//Check for next correction update 
IF fCurrentColumnPos + _fColumnsToPrecharge > nChargedColumns AND nChargedColumns <= sDefGridSettings.nGridSizeX THEN
  fCurrentPreCharge := fCurrentColumnPos + _fColumnsToPrecharge;
  IF bEnableDeformation THEN 
    // sync deformation points
    WHILE FLOOR(fCurrentPreCharge) > nChargedColumns AND nChargedColumns <= sDefGridSettings.nGridSizeX DO
      nAvailPoints := _pAttachedCt^.nAvailableGridPoints;
      IF nAvailPoints >= sDefGridSettings.nGridSizeY * (nChargedColumns+1) THEN // Complete column available?
        nAvailPoints_mem := 0;
        LogLvl(Lvl:=E_LogSeverity.Debug, Msg:=F_Concat2('Charge CG col: ',TO_STRING(nChargedColumns)));
        FOR nRow := 0 TO sDefGridSettings.nGridSizeY - 1 DO
          // get points
          IF _pAttachedCt^.getDeformationPoint(nCol:=nChargedColumns, nRow:=nRow, sPoint => sPoint) THEN
            // transfer the displacement into a correction
            sPoint.dx := sPoint.dx;   // nothing to change
            sPoint.dy := sPoint.dy;
            
            // apply PU corrections
            correctionUpdate(pPoint:=ADR(sPoint));
            
            // correction limitation
            correctionLimit(pPoint:=ADR(sPoint));
            
            // send point
            IF NOT fbPs.newGridPoint(sPoint:=sPoint) THEN
               LogError(Msg:='stream new point failed');
               gridUpdate:=FALSE;
               RETURN;
            END_IF
          ELSE
            LogError(Msg:='get new grid point failed');
            gridUpdate:=FALSE;
          END_IF
        END_FOR
        
        nChargedColumns := nChargedColumns + 1;
      ELSE
        IF nAvailPoints > nAvailPoints_mem THEN // log once or after every update of new available poinst
          LogError(Msg:='point column expected but not available');
        END_IF
        nAvailPoints_mem := nAvailPoints;
        gridUpdate:=FALSE;
        RETURN;
      END_IF 
    END_WHILE
  ELSE
    // send points with no deformation
    FOR nRow := 0 TO sDefGridSettings.nGridSizeY - 1 DO
        MEMSET(destAddr:=ADR(sPoint), fillByte:=0, n:=SIZEOF(sPoint));
        sPoint.col := TO_DINT(nChargedColumns);
        sPoint.row := TO_DINT(nRow);
        IF NOT fbPs.newGridPoint(sPoint:=sPoint) THEN
           LogError(Msg:='stream new point failed');
           gridUpdate:=FALSE;
           RETURN;
        END_IF
    END_FOR
    nChargedColumns := nChargedColumns + 1;
  END_IF
END_IF
END_METHOD

METHOD InitWorkerPrint : BOOL
VAR_INPUT
  pAdsPg                : POINTER TO ST_ADS_PG;       // pg ads reference (worker prints ads)
  iDefGridParamMediator : I_ParamMediator;            // for deformation settings
  fLimitCorrectionX     : LREAL;                      // correction limit in y (abs) [px]
  fLimitCorrectionY     : LREAL;                      // correction limit in y (abs) [px]
END_VAR
IF NOT bInitialized            THEN LogError('Base Worker not initialized! call init() before'); RETURN; END_IF
IF pAdspg = 0 THEN LogError('InitWorkerPrint: invalid parameter proviced'); RETURN; END_IF
IF iDefGridParamMediator = 0   THEN bInitialized := FALSE; LogError('Invalid parameter, no valid param mediator'); RETURN; END_IF

// Worker specific init
_pAdsPg := pAdsPg;
_iParamMediator := iDefGridParamMediator;

_fLimitCorrectionX := ABS(fLimitCorrectionX);
_fLimitCorrectionY := ABS(fLimitCorrectionY);

// Print Aggregate
fbPa.bSyncAfterDone := FALSE;
fbPa.init(iPcAdapter := fB_PcAdapter, iPsInterface := fbPs);
END_METHOD

METHOD mJobPause
END_METHOD

METHOD   mJobStart
VAR_INPUT
	sJobDef	: CalmarCompPrint.I_JobDefinition;
END_VAR
// Config workers static variables
_fCtSecurityReleasePos := F_MeterToSubPixel(fPosMeter:=sJobDef.fImageDepth/1000 + fC_MIN_SHEET_GAP, fResoSubPx:=_fPrintResolution*_fSubPxResolution);

IF NOT bWorkerEnable THEN RETURN; END_IF  // only if enabled

fbPa.jobStart();

_sCurrentImgDepth := sJobDef.fImageDepth/1000;
_bEndless := sJobDef.isEndless();

_bJobActive := TRUE;
END_METHOD

METHOD  mJobStop
VAR_INPUT
	sStatus	: CalmarCompPrint.I_JobStatus;
END_VAR
fbPa.jobStop();
_bJobActive := FALSE;
_bPaStarted := FALSE;
_bPaStartRequested := FALSE;
END_METHOD

METHOD mProduced
VAR_INPUT
	(* current progress*)
	sProgress	: CalmarCompPrint.I_JobProgress;
END_VAR
END_METHOD

METHOD RegisterGridCorrection : BOOL
VAR_INPUT
  iGridCorrection : I_GridPointCorrection;
END_VAR
VAR
  i : UDINT;
END_VAR
IF iGridCorrection = 0 THEN LogError('registerGridCorrection: ivalid interface, ignore'); RETURN; END_IF
IF nPointCorrections >= nC_NUM_POINTCORRECTIONS THEN LogError('registerGridCorrection: too many corrections registred, ignore'); RETURN; END_IF

nPointCorrections := nPointCorrections + 1;
iPointCorrections[nPointCorrections] := iGridCorrection;
END_METHOD

METHOD registerPc : BOOL
VAR_INPUT
  iNewPC : I_PC;
END_VAR
registerPc := fB_PcAdapter.registerPc(iNewPC := iNewPC);
END_METHOD

METHOD registerPh : BOOL
VAR_INPUT
    iPH : I_PH;
    iNewCG : I_Correction_Grid;   // correction grid interface
END_VAR
//Attach head to print station
IF iPH <> 0 THEN
  fbPs.registerCG(iNewPh:=iPH, iNewCG:=iNewCG);
END_IF
END_METHOD

METHOD PRIVATE sim
END_METHOD

METHOD PRIVATE updateWorkerPosition
VAR_INPUT
END_VAR
// Update only without attached container
IF _pAttachedCt = 0 THEN RETURN; END_IF

//Start offset update
IF _fPrintStartOffset <> (fPrintStartOffset + _iWorkerParams.fDetectToRefPos) THEN //Worker position changed
  _fPrintStartOffset := fPrintStartOffset + _iWorkerParams.fDetectToRefPos;
END_IF

//Worker position update
IF _fWorkerPosition <> (_fPrintStartOffset + (_fStartShiftOffset + _fStartShiftFactor * fMasterSpeed)) THEN   // Worker position changed (camera settings change)
  // WorkerPosition = PrintStart offset - pre-start offset
  fPosition := _fPrintStartOffset + (_fStartShiftOffset + _fStartShiftFactor * fMasterSpeed);
END_IF
END_METHOD

METHOD  work
VAR
  bDeformErr : BOOL;
  nDeformStep : E_DeformationStep;
END_VAR
IF _iWorkerParams = 0 OR _iParamMediator = 0 THEN F_Report_Error(ErrType:=EN_REPORT_ERROR_TYPE.Report_Error_0Pointer); RETURN; END_IF
bError := FALSE; nError := 0;

updateWorkerPosition();  // calculate and set worker position

SUPER^.work();

(*Print correction*)
fbDropSpeedComp(fMasterSpeed:=fMasterSpeed, fDropTravelDistance:=fPUElevation);


(*Update virtual encoder on all controller boards*)
fB_PcAdapter.setEncoderPos(nPrintPos);
fB_PcAdapter();

(*Call print aggregate*)
rTrigHwSync(CLK:=bHardwareSync); 
IF rTrigHwSync.Q THEN fbPa.sync(); END_IF   // external sync cmd
fbPa.bHold := bHardwareHold;                // external hw hold, NOTE: this stop the current print iPC.stop()
fbPa();

fBStartTimeout(IN:=_bPaStartRequested, PT := T#60MS);

IF _pAttachedCt <> 0 AND bWorkerEnable THEN // Work only with attached container
  
  // check for generic error
  IF _pAttachedCt^.bValid AND bHardwareHold THEN
    // abort during printing
    _pAttachedCt^.setError(ErrDef:=EC_Print.ecPaAbortHold, Src:=_pEcSrc^);
  END_IF

  // Grid update
  bDeformErr := _pAttachedCt^.getDeformationStatus(eDStep=>nDeformStep);
  IF NOT bDeformErr AND nDeformStep >= E_DeformationStep.gridStarted AND NOT _bForceDefGridOff THEN 
    IF NOT gridUpdate(bEnableDeformation:=TRUE) THEN
      _pAttachedCt^.AbortDeformation(sReason:='deformation point update failed', Src:=_pEcSrc^);
      //Release(iCT:=_pAttachedCt^);
    END_IF
  ELSE
    // not started or error already --> erase deformation points and send no correction points
    IF NOT gridUpdate(bEnableDeformation:=FALSE) THEN
      _pAttachedCt^.AbortDeformation(sReason:='deformation point update failed', Src:=_pEcSrc^);
      //Release(iCT:=_pAttachedCt^);
    END_IF
  END_IF

  // PA control
  IF _bPaStartRequested THEN
    IF fbPa.bPrinting THEN
      _bPaStarted := TRUE;
      _bPaStartRequested := FALSE;
    ELSIF fBStartTimeout.Q THEN //Stop print at timeout to make ready for next container
      _bPaStarted := FALSE;
      _bPaStartRequested := FALSE;
      fbPa.printStop();
      _pAttachedCt^.setError(ErrDef:=EC_Print.ecPaStartErr, Src:=_pEcSrc^);
      Release(_pAttachedCt^);
		END_IF
  ELSIF _bPaStarted THEN
    //Release container when all points have been processed
    IF fbPa.bDone OR fbPa.bStop THEN
      _bPaStarted := FALSE;
      Release(_pAttachedCt^);
    (*ELSIF fbpa.bError THEN
      _pAttachedCt^.setError(ErrDef:=EC_Print.ecPaPrintErr, Ident:=0);
      Release(_pAttachedCt^);*)
    ELSE
      // still printing (endless or not yet done)
      IF _bEndless AND nChargedColumns >= sDefGridSettings.nGridSizeX THEN
        // in endless release if grid was streamed
        {warning 'TODO: send real PrintLength _pAttachedCt^.bPrintLength'} 
        Release(_pAttachedCt^);
			END_IF
    END_IF 
	END_IF
END_IF  


// forward pa state to pg ads
IF _pAdsPg <> 0 THEN
  _pAdsPg^.aO_State := fbPa.aPaState;
  _pAdsPg^.lO_Error := nError; 
  _pAdsPg^.bO_Error := bError;
END_IF

// logging config
fbPa.LogLevel := LogLevel;
fB_PcAdapter.LogLevel := LogLevel;

sim();
END_METHOD

END_FUNCTION_BLOCK

// ---- POUs/Products/Print_Weu/Mark/FB_MarkDefinition.TcPOU
(*
  Holds Marks definition & current state.
*)
{attribute 'no_explicit_call' := 'do not call this POU directly'} 
FUNCTION_BLOCK FB_MarkDefinition EXTENDS T_NamedBase IMPLEMENTS I_MarkDefinition
VAR
  // marks
  // - mark list
  _nMarks : UDINT;          // number of registered (teached) marks
  sMarkDef : ARRAY[1..50] OF ST_MarkDefinition;   // teached marks
  // - border mark
  _bBorderMarkUsed : BOOL;   // a border mark was teached
  sSheetBorderEndMark : ST_MarkDefinition;  // internal mark created on edge of sheet (used for effective sheet length)
  
  // mark states
  _nMarksDetected : UDINT;  // number of detected marks
  _bSheetBorderDetected : BOOL;
  _fSubstrateLengthEffective      : LREAL;        // detected substrate length

  // internals
  nMaxMarks : UDINT;
  sLastStartMark : ST_MarkDefinition;       // sampled start mark (because first mark will be overwritten already by next sheet)
END_VAR

(*
  Definition of a mark.
  
   SqLength | TrLength -->
   |--------|--------
   |        |      /
   |        |    / -- center --
^  |        |  /
|  |--------|
| Height

Requirements:
  - StartMark has to be unique (minimal length > than max. length of Other marks)
  - Distance between Start and Endmark has to be bigger than length of StartMark + Minimal space
  - Mark has a minimum lenth, so the sensor can see the mark

*)

(*
  Ge minimum length of hte start mark.
*)
PROPERTY fMinLengthStartMark : LREAL
GET
IF _nMarks > 0 THEN
  fMinLengthStartMark := sMarkDef[1].fSqLength;
END_IF
END_GET
END_PROPERTY

(*
  Get a mark definition.
  nIdx= 1.._nMarks = registered marks
  nIdx= 0 - selects last mark 
  nIdx=-1 - selects border mark
  :returns: pointer to mark defintion or 0 if not found
*)
METHOD getMark : POINTER TO ST_MarkDefinition
VAR_INPUT
  nIdx : DINT; // mark index: 1.._nMarks, 0 = last (endMark) 
END_VAR
IF    nIdx = 0 THEN 
  getMark := ADR(sMarkDef[_nMarks]); // last mark (end or last)
ELSIF nIdx = -1 THEN
  IF _bBorderMarkUsed THEN
    getMark := ADR(sSheetBorderEndMark);  // sheet border mark
  END_IF  
ELSIF nIdx > 0 AND nIdx <= TO_DINT(_nMarks) THEN 
  getMark := ADR(sMarkDef[nIdx]);
ELSE 
  LogError(F_Concat2('Invalid mark requested, Idx=', TO_STRING(nIdx)));
END_IF
END_METHOD

METHOD Init : BOOL
VAR_INPUT
END_VAR
nMaxMarks := SIZEOF(sMarkDef) / SIZEOF(sMarkDef[1]);
ResetDefinition();
END_METHOD

(*Number of registered marks*)
PROPERTY nMarks : UDINT
GET
nMarks := _nMarks + SEL(_bBorderMarkUsed, 0, 1);
END_GET
END_PROPERTY

(*Number of detected marks*)
PROPERTY nMarksDetected : UDINT
GET
// number of detected marks + sheetborder if used
nMarksDetected := _nMarksDetected + SEL(_bBorderMarkUsed AND _bSheetBorderDetected, 0, 1);
END_GET
END_PROPERTY

PROPERTY pLastStartMark : POINTER TO ST_MarkDefinition
GET
pLastStartMark := ADR(sLastStartMark);
END_GET
END_PROPERTY

(*
  Register a mark to camera (teach).
  If mark.nId >= 0 then it will be a detectable mark.
  If mark.nId = -1 it will be the sheet-end border mark
*)
METHOD RegisterMark : BOOL
VAR_INPUT
  sMark : ST_MarkDefinition;
END_VAR
VAR
  pMark : POINTER TO ST_MarkDefinition;
END_VAR
IF sMark.nId = -1 THEN
  // - border mark
  _bBorderMarkUsed := TRUE;
  pMark := ADR(sSheetBorderEndMark);
  // copy mark data
  pMark^ := sMark;
  // view 
  pMark^.bShow := FALSE;
  pMark^.nMove := TO_DINT(_nMarks+1);
ELSE
  // - for all other teach marks
  IF _nMarks >= nMaxMarks THEN LogError('Number of marks exeeded, ignore'); RETURN; END_IF
  // we assume first mark is start mark, last mark is end mark (marks need to be registered in sorted order)
  // (TODO) otherwise add marks in a sorted way to list
  _nMarks := _nMarks + 1;
  pMark := ADR(sMarkDef[_nMarks]);
  // copy mark data
  pMark^ := sMark;

  // set id if not given
  IF pMark^.nId = 0 THEN pMark^.nId := TO_DINT(_nMarks); END_IF
  
  // view
  pMark^.bShow := TRUE;
  pMark^.nMove := TO_DINT(pMark^.nId-1);
  
  // checks
  IF _nMarks > 1 THEN   
    // -- start mark length requirement 
    IF pMark^.fSqLength + pMark^.fTrLength >= sMarkDef[1].fSqLength THEN 
      LogError(F_Concat5('RegisterMark: mark not unique, too long: ', TO_STRING(pMark^.fSqLength + pMark^.fTrLength), ' > ', TO_STRING(sMarkDef[1].fSqLength), ' of start min. length'));
    END_IF
  END_IF
END_IF  


// clear eventual mark state
MEMSET(destAddr:=ADR(pMark^.sState), 0, SIZEOF(ST_MarkState));

RegisterMark := TRUE;
END_METHOD

METHOD ResetDefinition
VAR
  i : UDINT;
END_VAR
ResetMarkStates();

_nMarks := 0;
_bBorderMarkUsed:=FALSE;

MEMSET(destAddr:=ADR(sMarkDef), fillByte:=0, SIZEOF(sMarkDef));
MEMSET(destAddr:=ADR(sLastStartMark), fillByte:=0, SIZEOF(sLastStartMark));
MEMSET(destAddr:=ADR(sSheetBorderEndMark), fillByte:=0, SIZEOF(sSheetBorderEndMark));
// prepare border point
sSheetBorderEndMark.nId := -1;
END_METHOD

(*
  Reset all registered marks
*)
METHOD ResetMarkStates
VAR
  i : UDINT;
END_VAR
// reset detected marks
_nMarksDetected := 0;
_bSheetBorderDetected := FALSE;
_fSubstrateLengthEffective := 0;
// reset mark state only
FOR i:=1 TO _nMarks DO
  MEMSET(destAddr:=ADR(sMarkDef[i].sState), 0, SIZEOF(ST_MarkState));
END_FOR
//MEMSET(destAddr:=ADR(sLastStartMark.sState), 0, SIZEOF(ST_MarkState));
MEMSET(destAddr:=ADR(sSheetBorderEndMark.sState), 0, SIZEOF(ST_MarkState));
END_METHOD

METHOD saveMark : BOOL
VAR_INPUT
  pMark : POINTER TO ST_MarkDefinition;
END_VAR
IF pMark = 0 THEN RETURN; END_IF

// sample start mark
IF pMark^.nId = 1 THEN 
  sLastStartMark := pMark^;           // save start mark as backup
  sMarkDef[pMark^.nId] := pMark^;     // save in teached mark table
  _nMarksDetected := _nMarksDetected + 1;
  saveMark := TRUE;

ELSIF pMark^.nId = -1 AND _bBorderMarkUsed THEN
  sSheetBorderEndMark := pMark^;     // save sheet border point
  _bSheetBorderDetected := TRUE;
  saveMark := TRUE;
  
ELSIF pMark^.nId > 1 AND pMark^.nId <= TO_DINT(_nMarks) THEN
  sMarkDef[pMark^.nId] := pMark^;     // save in teached mark table
  _nMarksDetected := _nMarksDetected + 1;
  saveMark := TRUE;  
  
ELSE
  LogError(F_Concat3('saveMark: mark with id=', TO_STRING(pMark^.nId), ' not available'));
END_IF
END_METHOD

END_FUNCTION_BLOCK

// ---- POUs/Products/Print_Weu/Mark/FB_MarkDetection.TcPOU
(*
  Detects Marks and generates StartTrigger based on one EL1252 timestamp input I/O.
  
  Additionally:
    - returns lateral offset (+/- in [m]) to center of detected marks.
    - manages & supervises mark sequence
    - is a CameraTrigger as well
    - supports simulation mode
  
  NOTE: 
    - a mark has always a rising and falling edge of the sensor (triangle)
    - center position is the middle of the triangular mark

*)
FUNCTION_BLOCK FB_MarkDetection EXTENDS T_NamedBase IMPLEMENTS I_StartPosDetect, I_CameraTrigger, I_Sim
VAR_INPUT
  (*EL1252*)
  bIKp_StartSensor          AT%I* : BOOL;            (*Sensor start trigger*)
  tIKp_TimeStampPos         AT%I* : T_DCTIME64;      (*TimeStamp Pos_Edge @EL1252*)
  tIKn_TimeStampNeg         AT%I* : T_DCTIME64;      (*TimeStamp Neg_Edge @EL1252*)

  // configuration
  bEnable                         : BOOL;            (*Enable start pos detection sensor*)
  bAutomaticMode                  : BOOL;            (*machine is in automatic mode *)
  nCurrentPos                     : DINT;            (*current position in Pulses/Subpixels*)
  fCurrentSpeed                   : LREAL;           (*actual speed of conveyor in [m/s]*)
  
  // Debug & Test
  bManualTrigger                  : BOOL;            // Manual start trigger
  bManualReset                    : BOOL;            // Manaul reset detection
END_VAR
VAR
  bInitOk                         : BOOL;           // fb initialized

  // config
  _fResolution                    : LREAL := 1;     // current used print resolution (dpi*SubPx)
  _pFbMarkDefinition              : POINTER TO FB_MarkDefinition;      // mark definition
  _iCamera                        : I_Camera;       // camera interface
  // settings                                    
  _bUseCameraTrigger              : BOOL;           // (cam specific setting) Generate camera trigger output
  _bUseCameraTriggerFeedback      : BOOL;           // (cam specific setting) Evaluate camera triggered feedback
  _bCamManualTeachMode            : BOOL;           // cam in manual teach mode
  _fSubstrateLength               : LREAL;          // Substrate length in [m] (should be repeat ength)
  _fTriggerDistance               : LREAL;          // Distance between Sensor and Trigger [m]
  _fTriggerLength                 : LREAL := 10;    // Length of trigger signal in ms, min. 3 bus cycles
  _iActiveCam                     : I_CameraTriggerDevice;  // active camera interface (set by Enable() on I_CameraTrigger)

  // sensor
  bSheetActive                    : BOOL;           (*sheet is scanning*)
  bSpeedValid                     : BOOL;           (*speed is valid*)
  bTriggerArmed                   : BOOL;           (*trigger is armed*)
  bCamValid                       : BOOL;           (*camera is valid*)
  bMarkValid                      : BOOL;           (*definition is valid marks&substrate*)
  
  // helper
  rfT_Enable                      : RF_TRIG;        // edge detection enable
  bResetMethods                   : BOOL;           (*Reset request for checkForMark() internals*)
  isStartMark                     : BOOL;
  isMarkError                     : BOOL;
  nMarkSelection                  : UDINT := 1;     (*Current selected mask to search*)
  pMarkSearch                     : POINTER TO ST_MarkDefinition;
  _fSubstrateLengthEffective      : LREAL;          // Substrate length in [m]
  
  // time calculations
  tNowDc                          : T_DCTIME64;     (* Get Current Timestamp (now)*)
  fCycleTime                      : LREAL;          (*Current calculated cycle time [s]*)
  
  // params
  _bStartTrig                     : BOOL;           // Start Trigger Edge
  _nX0                            : DINT;           // X0 Position [SubPx]
  _bValid                         : BOOL;           //
  
  // simulation & debug
  _bSimEnable                     : BOOL;           // simulation mode enabled
  _bVerbose                       : BOOL;           // verbose mode
  // view 
  nMarkXMoveScale                 : UDINT := 140;
END_VAR
VAR PERSISTENT
  bR_TerminateLast                : BOOL;           // Terminate sheet with last defined & detected mark
  bR_CreateBorderMark             : BOOL;           // Create a (virtual) mark at end-border of sheet
  nR_AreaMarkSensorOk             : INT := 10;      (*Area with the correct arrangement of the mark sensor [%]*)
END_VAR
VAR CONSTANT
  fC_InhibitSubstrateMargin       : LREAL := 0.010;   (*[m] decrease substrate for inhibit in*)
  fC_MinimalSpeed                 : LREAL := 0.010;   //[m/s]
  fC_MarkLengthMargin             : LREAL := 0.005;   // [m]
  fC_MaxSubstrateFactor           : LREAL := 1.025;   // factor which the sheet length can be max. longer
END_VAR

// check parameter
IF NOT bInitOk THEN RETURN; END_IF

// General calculations
bSpeedValid   := fCurrentSpeed > fC_MinimalSpeed;                // speed valid (ignore trigger if not moving)
bCamValid     := SEL(_iActiveCam<>0, FALSE, TRUE);               // camera valid (ignore trigger otherwise)
bMarkValid    := (_fSubstrateLength > 0 AND _pFbMarkDefinition^.nMarks > 0);
tNowDc        := F_GetCurDcTaskTime64();                         // current dc time (most accurate time stamp we have)
fCycleTime    := calcCycleTime(tCurrent:=tNowDc);                // calculate cycle time of this fb
bTriggerArmed :=  bCamValid AND bSpeedValid AND bEnable AND bMarkValid AND (bAutomaticMode OR _bCamManualTeachMode OR _bSimEnable);   // trigger

IF bCamValid THEN    // (not yet used) save dynamic changable settings
  _fTriggerDistance := _iActiveCam.fTriggerDistance;
  _fTriggerLength   := _iActiveCam.fTriggerPulseLength;
END_IF

_bValid := _bStartTrig := FALSE;    // default values (outputs and properties)

manualTrigger();     // handle manual trigger

// enable & reset
rfT_Enable(CLK:=bEnable);             // edge detection (or use bTriggerArmed)
IF rfT_Enable.RT OR rfT_Enable.FT OR bManualReset THEN Reset(); bManualReset:=FALSE; END_IF;
IF NOT bEnable THEN RETURN; END_IF    // do nothing if not enabled
IF NOT bTriggerArmed THEN RETURN; END_IF


// Work
// - detect marks
//   - detect missing marks (based on teach definition, type and a margin)
//   - maybe replace missing marks (trend or teach)
// - handle StartTrigger if StartMark rising edge
// - handle Mark detected position (y-correction)
// - save mark, keep tracking of detected marks, (error handling if some missed)
// - send mark to camera


(*State Machine ----------------------------------------------------------------*)
// select mark
pMarkSearch :=  _pFbMarkDefinition^.getMark(nIdx:=TO_DINT(nMarkSelection));
// search for mark
IF checkForMark(pMark:=pMarkSearch, bStartMark=>isStartMark, bErr=>isMarkError) THEN 

  IF _bVerbose THEN LogInfo(F_Concat6('found mark: Start=', SEL(isStartMark,'0','1'), ' Err=', SEL(isMarkError,'0','1'), ' ', strMark(pMark:=pMarkSearch))); END_IF  

  // searched start, found start (normal start)
  IF isStartMark AND nMarkSelection = 1 THEN
    IF _pFbMarkDefinition^.nMarks = 1 THEN 
      // only one mark --> TERMINATE + START
      // - start
      SheetStart(pMark:=pMarkSearch);
      IF bR_TerminateLast THEN SheetStop(nNewX0:=0); END_IF  // TERMINATE already after single mark scanned
    ELSE
      // more marks --> START + NEXT
      // - start
      SheetStart(pMark:=pMarkSearch);
      // - next
      nMarkSelection := nMarkSelection + 1;    // next mark
		END_IF

  // search other mark and found start mark (start abort)
  ELSIF isStartMark AND nMarkSelection > 1 THEN
    // terminate(abort) last
    IF nMarkSelection < _pFbMarkDefinition^.nMarks THEN
      LogError('New start mark before last mark detected, missed a mark?');
    END_IF 

    // terminate/abort with new --> TERMINATE + START
    // - start
    SheetStart(pMark:=pMarkSearch);
    
    nMarkSelection := nMarkSelection + 1;    // next mark

  // intermediate marks
  ELSIF NOT isStartMark AND nMarkSelection > 1 THEN
    // search and found other --> NEXT (ev. terminate)
    
    IF _pFbMarkDefinition^.nMarksDetected <= _pFbMarkDefinition^.nMarks THEN
      // - save mark
        _pFbMarkDefinition^.saveMark(pMark:=pMarkSearch);
      // - last mark?
      IF nMarkSelection = _pFbMarkDefinition^.nMarks THEN
        IF bR_TerminateLast THEN SheetStop(nNewX0:=0); END_IF
        nMarkSelection := 1;
      ELSE
        nMarkSelection := nMarkSelection + 1;    // next mark
      END_IF 
    END_IF
	END_IF
END_IF


// outputs
// _bStartTrig := // set in SheetStart
// _nX0 :=  // set in SheetStart
_bValid := TRUE;

(*
  Check if mark was detected properly and type matches.
  :returns:  TRUE if in OK area
*)
METHOD PRIVATE analizeMark : BOOL
VAR_INPUT
  pMark           : POINTER TO ST_MarkDefinition;     // mark to search for
  fRealMarkLength : LREAL;                            // real detected mark length [m]
END_VAR
VAR_OUTPUT
  bStartMark : BOOL;     // a start mark was detected
END_VAR
IF pMark = 0 THEN RETURN; END_IF
IF pMark^.fHeight = 0 OR pMark^.fTrLength = 0 THEN analizeMark := TRUE; RETURN; END_IF

(*
  Sensor should aligned to the middle of the sensor (fI_MarkHeight / 2)
  With the difference OF the measured length TO the normal lenght, the fO_LateralOffset can be calculated
  invert in CASE OF wrong mirrored marks 
*)


{warning 'TODO: check if this is correct based on defined mark type'}
pMark^.sState.fLengthReal := fRealMarkLength;
// - dx  (based on sheet begin) dx = current mark position - teached mark position
pMark^.sState.dx := getMarkDistanceEffective(pMark:=pMark) - pMark^.fPosX;
  
// - dy 
pMark^.sState.dy := (pMark^.sState.fLengthReal * (pMark^.fHeight / 2 ) / ((pMark^.fTrLength / 2) + pMark^.fSqLength)) - (pMark^.fHeight / 2 );
IF pMark^.bInvertedX THEN
  pMark^.sState.dy := -1*pMark^.sState.dy;    
END_IF

// check position qualitiy
pMark^.sState.bInArea := FC_COMPARE_RANGE_PERCENT( 
                                       fI_ValueSet := (pMark^.fHeight / 2)
                                     , fI_ValueActual  := (pMark^.fHeight / 2) + pMark^.sState.dy
                                     , fI_RangePercent := nR_AreaMarkSensorOk);

// type of mark
bStartMark := (fRealMarkLength >= _pFbMarkDefinition^.fMinLengthStartMark);
pMark^.sState.bSet := TRUE;

analizeMark := pMark^.sState.bSet;
END_METHOD

PROPERTY bManualTeach : BOOL
GET
bManualTeach := _bCamManualTeachMode;
END_GET
SET
_bCamManualTeachMode := bManualTeach;
END_SET
END_PROPERTY

{attribute 'monitoring' := 'call'}
(*Simulation is enabled set/get*)
PROPERTY bSimEnable : BOOL
GET
bSimEnable := _bSimEnable;
END_GET
SET
_bSimEnable := bSimEnable;
END_SET
END_PROPERTY

(*
  A new container detected.
  NOTE: a pulse only
*)
PROPERTY bStartTrig : BOOL
GET
bStartTrig := _bStartTrig;
END_GET
END_PROPERTY

(*
  A valid container detected.
*)
PROPERTY bValid : BOOL
GET
bValid := _bValid;
END_GET
END_PROPERTY

METHOD PRIVATE calcCycleTime : LREAL
VAR_INPUT
  tCurrent : T_DCTIME64;
END_VAR
VAR_INST
  tLastTimeStamp : T_DCTIME64 := 0;
END_VAR
calcCycleTime := (TO_LREAL(tCurrent) - TO_LREAL(tLastTimeStamp)) * 1E-9;
tLastTimeStamp  := tCurrent;  // memory timestamp
END_METHOD

(*
  Poll for sensor triggers and marks.
  :return: true if a mark was detected
*)
METHOD PRIVATE checkForMark : BOOL
VAR_INPUT
  pMark : POINTER TO ST_MarkDefinition;             // mark to search for
END_VAR
VAR_OUTPUT
  bErr : BOOL;
  bStartMark : BOOL;     // a start mark was detected
END_VAR
VAR_INST
  rfT_StartSensor                 : RF_TRIG;        // edge detection start trigger
  tRisingEdge, tFallingEdge       : T_DCTIME64;     // detected edges
  nRisingPos, nFallingPos         : DINT;           // detected [SubPx] pos
  fMarkDuration                   : LREAL;
  fDeltaDistance                  : LREAL;          (*Distance that the substrate moved between the detection and the treatment of the information [m]*)
   
  bMarkStartDetected              : BOOL;   // mark started
  bMarkEndDetected                : BOOL;   // marks end reached
  bDone   : BOOL;
  
  // (Todo) inhibit control
  bInhibitTrigger                 : BOOL;       (*inhibit sensor signals, TRUE=inhibit*)
  nInhibitSensorDistance          : DINT;       (*inhibit length in pulseto X0 [SubPx]*)
  bReleaseSensor                  : BOOL;       (*condition to send a stop trigger*)
END_VAR
IF pMark = 0 THEN RETURN; END_IF
IF bDone OR bResetMethods THEN   // reset methods internal states
  bMarkStartDetected := FALSE;
  bMarkEndDetected := FALSE;
  bInhibitTrigger := FALSE;
  bResetMethods := FALSE;
  bErr := FALSE;
  bDone := FALSE;
END_IF

IF _bSimEnable THEN 
  checkForMark := SimMarks(pMark:=pMark, bStartMark=>bStartMark);
  RETURN;
END_IF

rfT_StartSensor(CLK:=bIKp_StartSensor);   // edge detection

// -- rising edge detection
IF rfT_StartSensor.RT AND NOT bInhibitTrigger THEN
  tRisingEdge := tIKp_TimeStampPos;
  bMarkStartDetected := TRUE;
  
  IF bMarkStartDetected OR bMarkEndDetected THEN 
    LogError(F_Concat3('Rigsing trigger while already a ', SEL(bMarkStartDetected, 'falling', 'rising') ,' edge was detected'));
    bErr := TRUE;
    {warning 'TODO: implement a fallback in any case'}
  END_IF
  
 // before calculation with some compensation
(*
  // Calculate the original position in our position domain
  tCurrentTime  := F_GetCurDcTaskTime64();
  fL_CurrentTimeStamp  := (ULINT_TO_LREAL(tCurrentTime) - (nC_CurrentTimeStampComp * 1_000)) / 1_000_000.0; (*in ms*)
  fI_Sensor_TimeStamp := (ULINT_TO_LREAL(tRisingEdge) - (nC_SensorTimeStampComp  * 1_000)) / 1_000_000.0; (*in ms*)

  // Treatment of the information
  fDeltaDistance := (fL_CurrentTimeStamp - fI_Sensor_TimeStamp) * 0.001 * fCurrentSpeed;	(* Distance in pulses that the substrate has traveled between the sensor detection and the PLC treatment *)
  iL_DeltaPosition := FC_LREAL_TO_DINT(fDeltaDistance * (1 / (0.0254 / fI_Resolution)));  (*1/1px*)	(* Travel of the substrate between the time of acquisition and the time of treatment *)
  nOffset_X0       := nCurrentPos - iL_DeltaPosition;	(* Position where the sheet has been detected *)
*)

  // like DMAX
  fDeltaDistance := UINT64_TO_LREAL(UInt64Sub64(ULINT_TO_ULARGE(tNowDc), ULINT_TO_ULARGE(tRisingEdge))) * 1E-9 * fCurrentSpeed;
  nRisingPos := nCurrentPos - F_MeterToSubPixel(fPosMeter:=fDeltaDistance, fResoSubPx:=_fResolution);    (*Position where the sheet has been detected in [SubPx]*) 
END_IF;


// -- falling edge detection
IF rfT_StartSensor.FT AND NOT bInhibitTrigger THEN
  // falling edge
  tFallingEdge := tIKn_TimeStampNeg;
  bMarkEndDetected := TRUE;
  
  fDeltaDistance := UINT64_TO_LREAL(UInt64Sub64(ULINT_TO_ULARGE(tNowDc), ULINT_TO_ULARGE(tFallingEdge))) * 1E-9 * fCurrentSpeed;
  nFallingPos := nCurrentPos - F_MeterToSubPixel(fPosMeter:=fDeltaDistance, fResoSubPx:=_fResolution);    (*Position where the sheet has been detected in [SubPx]*) 

  IF NOT bMarkStartDetected THEN 
    LogError('Missing rigsing trigger edge before falling edge');
    bErr := TRUE;
  END_IF

ELSIF bMarkStartDetected AND (nCurrentPos - nRisingPos) > (nRisingPos + F_MeterToSubPixel(fPosMeter:=pMark^.fTrLength + pMark^.fSqLength + fC_MarkLengthMargin, fResoSubPx:=_fResolution)) THEN
  // Expected falling edge missed
  LogWarning('Mark end missed');
  nFallingPos := nRisingPos + F_MeterToSubPixel(fPosMeter:=pMark^.fTrLength/2+pMark^.fSqLength, fResoSubPx:=_fResolution);
  bMarkEndDetected := TRUE;
  pMark^.sState.bMissed := TRUE;
  
END_IF;


{warning 'TODO: check if mark was missed and then analyze and send it without .bSet (missed (intermediate)mark)'}

// -- mark evaluation
IF bMarkStartDetected AND bMarkEndDetected THEN
  // mark finished
  
  // - define mark
  pMark^.sState.nPosXReal := nRisingPos;  // save detected mark pos
  fMarkDuration    := (ULINT_TO_LREAL(tFallingEdge) - ULINT_TO_LREAL(tRisingEdge));		// Calculate how long the signal was ON
  
  // check mark & calculate offsets
  IF analizeMark( pMark:=pMark, fRealMarkLength:=fMarkDuration * fCurrentSpeed * 0.000_000_001, bStartMark => bStartMark ) THEN
    checkForMark := TRUE;
  ELSE
   bErr := TRUE;  // invalid mark detected
	END_IF
  
  bDone := TRUE;   // done, reset states

ELSIF bErr THEN
  bDone := TRUE;
END_IF
END_METHOD

METHOD Disable : BOOL
_iActiveCam := 0;
Disable := TRUE;
END_METHOD

METHOD Enable : BOOL
VAR_INPUT
	iCam	                    : I_CameraTriggerDevice;
  bUseCameraTrigger         : BOOL; //Generate camera trigger
  bUseCameraTriggerFeedback : BOOL; //Use feedback as trigger?
END_VAR
IF iCam = 0 THEN
  Enable := FALSE;
  LogError('setCam failed: invalid reference');
ELSE
  _iActiveCam := iCam;
  Enable     := TRUE;

  // save constant settings
  _bUseCameraTrigger := bUseCameraTrigger;
  _bUseCameraTriggerFeedback := bUseCameraTriggerFeedback;
  
  IF _bUseCameraTrigger OR _bUseCameraTriggerFeedback THEN
    LogWarning('Enable: Camera Trigger output/feedback not yet supported');
	END_IF
END_IF;
END_METHOD

(*
  Get X0 from detected start mark
*)
METHOD PRIVATE getLastX0 : DINT
VAR
  pLastStartMark : POINTER TO ST_MarkDefinition;
END_VAR
pLastStartMark := _pFbMarkDefinition^.pLastStartMark;

IF pLastStartMark <> 0 THEN
  getLastX0 := pLastStartMark^.sState.nPosXReal - F_MeterToSubPixel(fPosMeter:=pLastStartMark^.fPosX, fResoSubPx:=_fResolution);
END_IF
END_METHOD

(*
  Calculate effective distance of mark to X0 [m]
*)
METHOD PRIVATE getMarkDistanceEffective : LREAL
VAR_INPUT
  pMark : POINTER TO ST_MarkDefinition;
END_VAR
VAR
  pFirstMark : POINTER TO ST_MarkDefinition;
END_VAR
IF pMark = 0 THEN RETURN; END_IF

IF pMark^.nId = 1 THEN 
  getMarkDistanceEffective := pMark^.fPosX;
ELSE
  pFirstMark := _pFbMarkDefinition^.getMark(nIdx:=1);
  IF pFirstMark <> 0 THEN
    // real distance between this mark and start mark + fPosX of start mark
    getMarkDistanceEffective := pFirstMark^.fPosX + F_SubPixelToMeter(lPosSubPx:=pMark^.sState.nPosXReal - pFirstMark^.sState.nPosXReal, fResSubPx:=_fResolution);
  END_IF
END_IF
END_METHOD

METHOD Init
VAR_INPUT
  fPrintResolution      : LREAL := 600;         // print(head) resolution in [dpi]
  fSubPxResolution      : LREAL := 32;          // SubPixel resolution [SubPx], resolution factor (fI_PrintResolution*fI_SubPxResolution=>Output resolution)
  pFbMarkDefinition     : POINTER TO FB_MarkDefinition;
END_VAR
IF fPrintResolution = 0 OR fSubPxResolution = 0 OR pFbMarkDefinition = 0 THEN LogError('Init: invalid parameter'); RETURN; END_IF

_fResolution := fPrintResolution * fSubPxResolution;
_pFbMarkDefinition:= pFbMarkDefinition;

Reset();
bInitOk := TRUE;
END_METHOD

METHOD PRIVATE manualTrigger : BOOL
VAR_INST
  rfTrig_ManuTrigger : RF_TRIG;
END_VAR
rfTrig_ManuTrigger(CLK:=bManualTrigger);

IF rfTrig_ManuTrigger.RT THEN
  LogWarning('manualTrigger not yet implemented');
END_IF

manualTrigger := rfTrig_ManuTrigger.RT;
END_METHOD

(*Print mark position (bit coded)*)
  (*Bit 0: no mark*)
  (*Bit 1: mark on drive side*)
  (*Bit 2: mark in center range*)
  (*Bit 3: mark on control side*)
PROPERTY nPrintMarkPosBits : WORD
GET
{warning 'TODO: implement'}
(*Print mark position (bit coded)*)
  (*Bit 0: no mark*)
  (*Bit 1: mark on drive side*)
  (*Bit 2: mark in center range*)
  (*Bit 3: mark on control side*)
nPrintMarkPosBits := 0;
END_GET
END_PROPERTY

(*
  Detected start position X0 (absolute) in [SubPx].
*)
PROPERTY nStartPositionX0 : DINT
GET
nStartPositionX0 := _nX0;
END_GET
END_PROPERTY

(*
  Reset internal state and all marks
*)
METHOD Reset
IF NOT bInitOk THEN RETURN; END_IF

_bValid := FALSE;
_bStartTrig := FALSE;
nMarkSelection := 1; // start mark

// reset camera (release if one is selected)
IF bSheetActive THEN
  IF _iActiveCam <> 0 THEN _iActiveCam.CamTriggerDone(); END_IF   // notify an done/abort
END_IF
_pFbMarkDefinition^.ResetMarkStates();  // reset detected marks
bSheetActive := FALSE;
bResetMethods := TRUE;        // reset checkForMark() state machine
END_METHOD

METHOD SetSubstrateLength
VAR_INPUT
  fSubstrateLength : LREAL;
END_VAR
IF NOT bInitOk THEN RETURN;END_IF;

(*reduced by margin (for endless mode with potential smaller printed repetition)*)
_fSubstrateLength := fSubstrateLength;
//_nSubstrateLength := F_MeterToSubPixel(fPosMeter:=_fSubstrateLength, fResoSubPx:=_fResolution);
END_METHOD

METHOD PRIVATE SheetStart
VAR_INPUT
  pMark : POINTER TO ST_MarkDefinition;
END_VAR
VAR
  sMarkBackup : ST_MarkDefinition;
END_VAR
_nX0 := pMark^.sState.nPosXReal - F_MeterToSubPixel(fPosMeter:=pMark^.fPosX, fResoSubPx:=_fResolution);
_bStartTrig := TRUE;

// (force) terminate a sheet
IF bSheetActive THEN 
  IF _bVerbose THEN LogInfo(F_Concat2('Terminate sheet with new Start Mark', '')); END_IF
  sMarkBackup := pMark^;   // push 
  SheetStop(nNewX0:=_nX0);
  pMark^:= sMarkBackup;    // pop
END_IF

IF _bVerbose THEN LogInfo(F_Concat2('SheetStart at X0=', TO_STRING(_nX0))); END_IF

// save (start) mark
_pFbMarkDefinition^.saveMark(pMark:=pMark);

// trigger camera
IF _iActiveCam<>0 THEN _iActiveCam.CamTrigger(bOk:=TRUE, nPos:=_nX0, nPosDeviation:=0); END_IF

bSheetActive := TRUE;
END_METHOD

METHOD PRIVATE SheetStop
VAR_INPUT
  nNewX0 : DINT;   // new detected X0
END_VAR
VAR
  pLastMark : POINTER TO ST_MarkDefinition;
  pBorderMark : POINTER TO ST_MarkDefinition;
  fD : LREAL;
  fSLen : LREAL;
  nDetectedX0 : DINT;
END_VAR
// - terminate
IF _bVerbose THEN LogInfo(F_Concat2('SheetStop()', '')); END_IF

fSLen := _fSubstrateLength;  // (default) original length

// calculate effective sheet length
nDetectedX0 := getLastX0();   // get sampled X0
IF nNewX0 <> 0 AND nDetectedX0 <> 0 THEN
  // real diff between two starts
  fD := F_SubPixelToMeter(lPosSubPx:=nNewX0 - nDetectedX0, fResSubPx:=_fResolution);
  IF fD < (_fSubstrateLength * fC_MaxSubstrateFactor) THEN
    fSLen := fD;
  END_IF 
ELSIF nNewX0 = 0 AND _pFbMarkDefinition^.nMarksDetected > 1 THEN
  // calculate based on last detected mark (a strech factor)
  pLastMark:= _pFbMarkDefinition^.getMark(nIdx:=0);     // get last available mark
  fD := getMarkDistanceEffective(pMark:=pLastMark); 
  fSLen := (pLastMark^.fPosX/SEL(fD<>0, pLastMark^.fPosX, fD)) * _fSubstrateLength; // estimate real length with last mark
END_IF
_fSubstrateLengthEffective := fSLen;


// set a (virtual) sheet border point (if activated)
pBorderMark := _pFbMarkDefinition^.getMark(nIdx:=-1);
IF bR_CreateBorderMark AND pBorderMark <> 0 THEN
  pBorderMark^.sState.bSet      := TRUE;
  pBorderMark^.fPosX            := _fSubstrateLength;
  pBorderMark^.fPosY            := 0;
  pBorderMark^.sState.dx        := _fSubstrateLengthEffective - _fSubstrateLength;
  pBorderMark^.sState.dy        := 0;
  pBorderMark^.sState.nPosXReal := SEL(nNewX0=0, nNewX0, nDetectedX0 + F_MeterToSubPixel(fPosMeter:=_fSubstrateLengthEffective, fResoSubPx:=_fResolution) );
  // no size information
  _pFbMarkDefinition^.saveMark(pMark:=pBorderMark);
END_IF


IF _iActiveCam<>0 THEN _iActiveCam.CamTriggerDone(); END_IF 
_pFbMarkDefinition^.ResetMarkStates();

bSheetActive := FALSE;
END_METHOD

METHOD PRIVATE SimMarks : BOOL
VAR_INPUT
  pMark : POINTER TO ST_MarkDefinition;
END_VAR
VAR_OUTPUT
  nX0 : DINT;
  bStartMark : BOOL;
END_VAR
VAR_INST
  bMarkOn : BOOL;
  nMarkStarted : DINT;
  fStartMarkOffset : LREAL;
  nLastStartMark : DINT;  // last detected start mark
  tTon_Mark : TON;
  rand : DRAND;
  rlrand : LREAL;
  l : DINT;
END_VAR
IF pMark = 0 THEN RETURN; END_IF

// when sim enabled AND auto-trigger then create a StartMark after every sheet/repeate length
//  then generate every following intermediate mark with a given length

IF NOT bMarkOn THEN  // start new mark
  // create rising edge
  IF pMark^.nId = 1 THEN
    // wait for next StartPosition
    IF F_SubPixelToMeter(lPosSubPx:=nCurrentPos - nLastStartMark, fResSubPx:=_fResolution) >= _fSubstrateLength THEN
      nLastStartMark := nCurrentPos;      // save start mark pos
      fStartMarkOffset := pMark^.fPosX;   // save start mark displacement from X0
      pMark^.sState.nPosXReal := nCurrentPos;  // save rising edge
      nMarkStarted := nCurrentPos;
      l := F_MeterToSubPixel(fPosMeter:=pMark^.fSqLength + (pMark^.fTrLength/2), fResoSubPx:=_fResolution); // mark length
      bMarkOn := TRUE;
    END_IF
	ELSE
    // wait for next mark position
    IF F_SubPixelToMeter(lPosSubPx:=nCurrentPos - nLastStartMark, fResSubPx:=_fResolution) >= pMark^.fPosX - fStartMarkOffset THEN
      pMark^.sState.nPosXReal := nCurrentPos;  // save rising edge
      nMarkStarted := nCurrentPos;
      l := F_MeterToSubPixel(fPosMeter:=pMark^.fSqLength + (pMark^.fTrLength/2), fResoSubPx:=_fResolution); // mark length
      bMarkOn := TRUE;
		END_IF
  END_IF
  
ELSE
  // create falling edge
  IF (nCurrentPos - nMarkStarted) > l THEN
    rand(Seed:=13, Num=>rlrand);  // TODO: find a right scale 
    analizeMark(pMark:=pMark, fRealMarkLength:=F_SubPixelToMeter(lPosSubPx:=nCurrentPos - nMarkStarted, fResSubPx:=_fResolution));
    bMarkOn := FALSE;
    If pMark^.nId = 1 THEN bStartMark := TRUE; END_IF
    SimMarks := TRUE;    // mark done
  END_IF
END_IF
END_METHOD

METHOD strMark : T_MaxString
VAR_INPUT
  pMark : POINTER TO ST_MarkDefinition;
END_VAR
VAR_INST
  fbStrFormat : FB_FormatString;
END_VAR
VAR
  IdFormatted : STRING;
END_VAR
fbStrFormat(sFormat:='%.2d', arg1:=F_DINT(pMark^.nId), sOut=>IdFormatted);
strMark := F_Concat6(
  F_Concat2('Id:',   IdFormatted),
  F_Concat2(' Set:', SEL(pMark^.sState.bSet,'0','1')),
  F_Concat2(' posX:', LREAL_TO_FMTSTR( pMark^.fPosX, 4, TRUE )),
  F_Concat2(' posY:', LREAL_TO_FMTSTR( pMark^.fPosY, 4, TRUE )),
  F_Concat2(' dx:', LREAL_TO_FMTSTR( pMark^.sState.dx, 4, TRUE )),
  F_Concat2(' dy:', LREAL_TO_FMTSTR( pMark^.sState.dy, 4, TRUE )),
);
END_METHOD

END_FUNCTION_BLOCK

// ---- POUs/Products/Print_Weu/Mark/FB_MarkCamera_WEU.TcPOU
(*
  Mark camera system on WEU machine
  1 mark sensor (optional: reverse mode - roll printed in reversed direction, sensor moved to other side)
*)
FUNCTION_BLOCK FB_MarkCamera_WEU EXTENDS FB_CameraBase 
VAR
  // config
  _iMarkDefinition          : I_MarkDefinition;     // link to detection logic (get points, teach points)
  
  // sample & delay of states
  Dly_Ton                       : TON;      // delay timer
  Dly_CamTrigger_Request        : BOOL;     // delayed CamTrigger() call request
  Dly_CamTrigger_bOk            : BOOL;     // delayed CamTrigger() parameter
	Dly_CamTrigger_nPos           : DINT;     // delayed CamTrigger() parameter
  Dly_CamTrigger_nPosDeviation  : DINT;     // delayed CamTrigger() parameter
  // teach info
  _bTeachOk                     : BOOL;
  _nTeachedPoints               : UDINT;
  // delay
  //  time or position
  
END_VAR

IF NOT _bInitialized THEN RETURN; END_IF

// The detection work is done in FB_MarkDetection
// This FB just uses(receives) the marks from the external implementation
// - Receives events CamTrigger & CamTriggerDone from MarkDetection
// - Get current marks and send them to the iCameraSink

IF _bSimulate THEN sim_update(); END_IF

Dly_Ton(IN:=Dly_CamTrigger_Request, PT:=T#4MS);  // deleay CamTrigger so CT will be for sure attached CameraWorker and Worker has enought time to see the CameraDone status
IF Dly_Ton.Q THEN Dly_CamTrigger_Request := FALSE;
  SUPER^.CamTrigger(bOk:=Dly_CamTrigger_bOk, nPos:=Dly_CamTrigger_nPos, nPosDeviation:=Dly_CamTrigger_nPosDeviation);
END_IF

IF _bCamTriggerStarted THEN
  sendCamPoints();
END_IF

METHOD CamTrigger
VAR_INPUT
  bOk             : BOOL;     // trigger is ok
	nPos            : DINT;     // camera triggered position
  nPosDeviation   : DINT;     // camera started deviation
END_VAR
IF NOT _bInitialized THEN RETURN; END_IF

(* 
  delay CamTrigger()
  Needed because in endless mode the Sheet-End is potentially already the next start mark
  and the CameraWorker would miss the CameraDone status (CameraTriggerDone()-->CameraTrigger() within same cycle
*)
Dly_CamTrigger_Request := TRUE;
Dly_CamTrigger_bOk := bOk;
Dly_CamTrigger_nPos := nPos;
Dly_CamTrigger_nPosDeviation := nPosDeviation;
//do after timeout in body: SUPER^.CamTrigger(bOk:=bOk, nPos:=nPos, nPosDeviation:=nPosDeviation);

_bTeachOk := (_iMarkDefinition.nMarks > 0);
_nTeachedPoints := _iMarkDefinition.nMarks;
END_METHOD

METHOD CamTriggerDone
IF NOT _bInitialized THEN RETURN; END_IF

// stream lasting points to Worker Camera
IF _bCamTriggerStarted THEN
  sendCamPoints();
END_IF

sendBorderPoint();

SUPER^.CamTriggerDone();
END_METHOD

{attribute 'monitoring':='call'}
PROPERTY eCameraMode : E_CameraMode
GET
eCameraMode := _eCameraMode;
IF _eCameraMode = E_CameraMode.Auto THEN
  eCameraMode := E_CameraMode.Live;
END_IF
END_GET
END_PROPERTY

PROPERTY eDeviceType : E_CameraDevice
GET
eDeviceType := E_CameraDevice.PrintMark;
END_GET
END_PROPERTY

METHOD GetCamStatus : BOOL
VAR_OUTPUT
  bConnectionOK  : BOOL;    // Camera connected
  bTeachOk       : BOOL;    // Teach successful
  nTeachedPoints : UDINT;   // Teached points for this job
  nScannedPoints : UDINT;   // Scanned points on current sheet
  bCamStarted    : BOOL;    // Camera trigger is active, cam started
  bCamDone       : BOOL;    // Camera finished on last CT
  bErrors        : ARRAY[1..GVL_Camera.nC_NbCamErrors] OF BOOL;  // generic error flag list
END_VAR
IF _iMarkDefinition = 0 THEN RETURN; END_IF

bConnectionOK  := TRUE;
bTeachOk       := _bTeachOk;
nTeachedPoints := _nTeachedPoints;
nScannedPoints := _nRxCamPoints;
bCamStarted    := _bCamTriggerStarted;
bCamDone       := _bCamTriggerDone;

GetCamStatus := bConnectionOK AND bTeachOk;   // camera ready
END_METHOD

METHOD InitMarkCamera
VAR_INPUT
  nPrintUnitResolution         : UDINT;    (*printhead pixel resolution [dpi]*)
  nPrintUnitSubPx              : UDINT;    (*print unit subPixel resolution [SubPx]*)
  iCameraTrigger               : I_CameraTrigger;
  iMarkDefinition              : I_MarkDefinition;  // mark detection fb
END_VAR
VAR
  bOK : BOOL;
END_VAR
SUPER^.Init( nPrintUnitResolution      := nPrintUnitResolution
           , nPrintUnitSubPx           := nPrintUnitSubPx
           , iCameraTrigger            := iCameraTrigger
           , bUseCameraTrigger         := FALSE
           , bUseCameraTriggerFeedback := FALSE);

IF NOT _bInitialized OR iMarkDefinition = 0 THEN LogError('Init: invalid parameter'); RETURN; END_IF

_iMarkDefinition := iMarkDefinition;

_bInitialized := TRUE;
END_METHOD

METHOD mJobStart : BOOL
IF eCameraMode <> E_CameraMode.NoCorrection THEN 
  TeachMarks();
END_IF
END_METHOD

METHOD PRIVATE sendBorderPoint
VAR
  pMark                     : POINTER TO ST_MarkDefinition;
END_VAR
pMark := _iMarkDefinition.getMark(nIdx:=-1);
IF pMark <> 0 AND_THEN pMark^.sState.bSet THEN
  // Send Mark (CamPoint) to CameraSink
  stCamPoint.x_ref := F_MeterToSubPixelReal(  fPosMeter:=pMark^.fPosX                                 (*[m]*)
                                            , fResoSubPx:=UDINT_TO_LREAL(_nPrintUnitResolution));     (*Result should be in pixels*)
  stCamPoint.y_ref := F_MeterToSubPixelReal( fPosMeter:=pMark^.fPosX                                  (*[m]*)
                                            , fResoSubPx:=UDINT_TO_LREAL(_nPrintUnitResolution));     (*Result should be in pixels*)
  stCamPoint.dx    := F_MeterToSubPixelReal( fPosMeter:=pMark^.sState.dx                              (*[m]*)
                                            , fResoSubPx:=UDINT_TO_LREAL(_nPrintUnitResolution));     (*Result should be in pixels*)
  stCamPoint.dy    := F_MeterToSubPixelReal( fPosMeter:=pMark^.sState.dy                              (*[m]*)
                                            , fResoSubPx:=UDINT_TO_LREAL(_nPrintUnitResolution));     (*Result should be in pixels*)
  stCamPoint.valid := pMark^.sState.bSet;

  IF _iCameraSink <> 0 THEN
    _iCameraSink.AddCamPoint(sDeformationPoint:=stCamPoint);
  END_IF
END_IF
END_METHOD

METHOD PRIVATE sendCamPoints
VAR
  i : UDINT;
  pMark : POINTER TO ST_MarkDefinition;
END_VAR
WHILE _nRxCamPoints < _iMarkDefinition.nMarksDetected DO
  
  pMark := _iMarkDefinition.getMark(nIdx:=TO_DINT(_nRxCamPoints+1));
  IF pMark <> 0 THEN
    // Send Mark (CamPoint) to CameraSink
    stCamPoint.x_ref := F_MeterToSubPixelReal(  fPosMeter:=pMark^.fPosX                                 (*[m]*)
                                              , fResoSubPx:=UDINT_TO_LREAL(_nPrintUnitResolution));     (*Result should be in pixels*)
    stCamPoint.y_ref := F_MeterToSubPixelReal( fPosMeter:=pMark^.fPosY                                  (*[m]*)
                                              , fResoSubPx:=UDINT_TO_LREAL(_nPrintUnitResolution));     (*Result should be in pixels*)
    stCamPoint.dx    := F_MeterToSubPixelReal( fPosMeter:=pMark^.sState.dx                              (*[m]*)
                                              , fResoSubPx:=UDINT_TO_LREAL(_nPrintUnitResolution));     (*Result should be in pixels*)
    stCamPoint.dy    := F_MeterToSubPixelReal( fPosMeter:=pMark^.sState.dy                              (*[m]*)
                                              , fResoSubPx:=UDINT_TO_LREAL(_nPrintUnitResolution));     (*Result should be in pixels*)
    stCamPoint.valid := pMark^.sState.bSet;
  
    IF _iCameraSink <> 0 THEN
      _iCameraSink.AddCamPoint(sDeformationPoint:=stCamPoint);
    END_IF
  ELSE
    LogWarning(F_Concat2('Requested mark not found, mark Idx=', TO_STRING(_nRxCamPoints+1)));
  END_IF
  
  _nRxCamPoints := _nRxCamPoints + 1;   // next mark
END_WHILE
END_METHOD

(*
  Set mode to camera.
  :return: TRUE if success
*)
METHOD setCameraMode : BOOL
VAR_INPUT
  eCameraMode : E_CameraMode;
END_VAR
IF eCameraMode = E_CameraMode.Auto OR
   eCameraMode = E_CameraMode.NoCorrection OR
   eCameraMode = E_CameraMode.Live
   //eCameraMode = E_CameraMode.Trend 
THEN
   
  _eCameraMode := eCameraMode;  // set desired mode
  setCameraMode := TRUE;
ELSE
  LogError(F_Concat3('Camera mode=', TO_STRING(eCameraMode), ' not supported by camera'));
  _eCameraMode := E_CameraMode.NoCorrection;
END_IF
END_METHOD

METHOD PRIVATE sim_update
// Not implemented
END_METHOD

{attribute 'monitoring':='variable'}
PROPERTY sName : STRING
GET
sName := 'Printmarks';
END_GET
END_PROPERTY

(*
  Calculate marks (position, shape) and register to mark definition. 
*)
METHOD PRIVATE TeachMarks : BOOL
VAR_INPUT
END_VAR
VAR
  i : UDINT;
  spacing : LREAL := 0.08;  // mark spacing
  asq : LREAL := 0.002;     // sqare a length
  atr : LREAL := 0.008;     // triangle length (same h / l)
  numMarks : UDINT;
  xOfs : LREAL := 0.0023;
  yOfs : LREAL := 0.0023;
  
  sNewMark : ST_MarkDefinition;
END_VAR


// TODO: this is only a reference caluclation for simulation, please adpat after definition by STAG
//       ...
IF _iMarkDefinition = 0 THEN RETURN; END_IF

_iMarkDefinition.ResetDefinition();

numMarks := TO_UDINT((_fSubstrateLength-2*xOfs) / spacing); //  // TO_UDINT(FLOOR(_fSubstrateLength / spacing);)
IF numMarks = 0 THEN numMarks := 1; END_IF   // at least one mark

// calculate position
FOR i:=1 TO numMarks DO
  sNewMark.fHeight := atr;
  sNewMark.fTrLength := atr;
  sNewMark.fSqLength := SEL(i>1, asq+1.5*atr, asq);
  sNewMark.fPosX := xOfs+(i-1)*spacing;
  sNewMark.fPosY := yOfs;
  sNewMark.bInvertedX := FALSE;
  
  _iMarkDefinition.RegisterMark(sMark:=sNewMark);
END_FOR
END_METHOD

END_FUNCTION_BLOCK

// ---- POUs/Products/Print_Weu/FB_PrintModule_WEU_View.TcPOU
FUNCTION_BLOCK FB_PrintModule_WEU_View
VAR
  // helper
  bInit   : BOOL;
  
  // config
  _pModule : POINTER TO FB_PrintModule_WEU;
  _pPositioning : POINTER TO FB_PrintPositionDmax;
  
  // view selections
  nSelWorkerPrint : UDINT := 1;
  bShowDropSpeedSetup : BOOL;
  // hardware view
  bShowPhDetail : BOOL;
  nSelPhDetail : UDINT := 1;
  bShowPcDetail : BOOL;
  nSelPcDetail : UDINT := 1;
  
  // motion and position view
  bShowPositionDetail : BOOL;
  bMovingInd : BOOL;
  fSpeed  : LREAL;
  fbBlink_Moving : FB_BLINK;
  
  // debug view
  bShowDebugAndSim : BOOL;
  
  fbBlink_Printing : FB_BLINK;
  bBlinkPrint : BOOL;
  bPrintInd : ARRAY[1..GVL_WEU.nC_WorkerPrintPerPm] OF BOOL;
  t : TIME;
  zPos_PM : UDINT;
  i : UDINT;
END_VAR

VAR CONSTANT
  nC_MAX_WORKER_VIEWS : UINT := 10;
END_VAR

IF NOT checkConfig() THEN RETURN; END_IF    // check config

// -- show moving -----------------------
fSpeed := _pPositioning^.getSpeed();
IF LrealIsNaN(x:=fSpeed) THEN
  fSpeed := 0;
END_IF
t := LREAL_TO_TIME(1000-fSpeed*900);
fbBlink_Moving(bI_Enable:=SEL(fSpeed > 0, FALSE, TRUE), tI_Time:=t, bO_Out=>bMovingInd);

t := T#400MS;
fbBlink_Moving(bI_Enable:=TRUE, tI_Time:=t, bO_Out=>bBlinkPrint);
FOR i:=1 TO GVL_WEU.nC_WorkerPrintPerPm DO
  bPrintInd[i] := _pModule^.fbWorkerPrint[i].bPrinting AND bBlinkPrint;
END_FOR


// -- show pm module position
zPos_PM := SEL(_pModule^._pModuleMachineState^.bUnitInPrintPosition, 0, 40);

// -- show ph detail
nSelPhDetail := LIMIT(1, nSelPhDetail, _pModule^._nPh);
nSelPcDetail := LIMIT(1, nSelPcDetail, _pModule^._nPc);

METHOD checkConfig : BOOL
VAR_INPUT
END_VAR
VAR_INST
  _fX_m, _fY_m   : LREAL;
  _nX_px, _nY_px : DINT; 
END_VAR
VAR
  bOK : BOOL;
END_VAR
IF NOT bInit THEN RETURN; END_IF

checkConfig := TRUE;
END_METHOD

METHOD init : BOOL
VAR_INPUT
  pModule : POINTER TO FB_PrintModule_WEU;
  pPositioning : POINTER TO FB_PrintPositionDmax;
END_VAR
IF pPositioning = 0 OR pModule = 0 THEN RETURN; END_IF

_pModule := pModule;
_pPositioning := pPositioning;

bInit := TRUE;
END_METHOD

END_FUNCTION_BLOCK

// ---- POUs/Products/Print_Weu/FB_ModuleMaster.TcPOU
(*
  This fb is the master controller of modules.
  Like an interface handler/provider for Module to Main communiation
*)
FUNCTION_BLOCK FB_ModuleMaster EXTENDS T_NamedBase IMPLEMENTS I_ModuleMaster, I_DeformationHandler, I_WorkerParams
VAR_OUTPUT
  fMasterSpeed    : LREAL;    // master speed [m/s]
  nMasterPosition : DINT;     // master position [SubPx]
END_VAR
VAR
  bInit : BOOL;
  // references
  _pPU : POINTER TO FB_PU;    // PU access
  _pProdMngr : POINTER TO FB_ProdManager_DMAX;
  _iHwPool : I_HardwarePool;  // reference of all harware
    
  // global instances
  fBCTManagerMain : FB_CTManagerDefGrid;  
  
  // print modules
  _sModules : ARRAY[1..nC_MaxModules] OF POINTER TO FB_PrintModule_Base;  // all registered print modules
  _nModules : UDINT;          // number of registered print modules
  // - active module
  _pMasterModule : POINTER TO FB_PrintModule_Base;  // current selected master module
  _iMasterPos : I_PrintPosition; // current master position interface
  _iMasterStartPosDetect : I_StartPosDetect;
  
  // helper
  iNewCt : I_CT;
  pCT : POINTER TO FB_ContainerDefGrid;
  
  // view
  nViewPmSel : UDINT := 1;  // visu pm selection
  
END_VAR
VAR CONSTANT
  nC_MaxModules : UDINT := 8;
END_VAR

IF NOT bInit OR _pMasterModule = 0 THEN RETURN; END_IF

_iMasterPos := _pMasterModule^.iPrintPosition;
IF _iMasterPos <> 0 THEN
  nMasterPosition := _iMasterPos.getPosition();
  fMasterSpeed := _iMasterPos.getSpeed();
END_IF

// Create CT
_iMasterStartPosDetect := _pMasterModule^.iStartPos;
IF _iMasterStartPosDetect <> 0 AND_THEN _iMasterStartPosDetect.bStartTrig AND _iMasterStartPosDetect.bValid THEN
  // create new CT
  iNewCt := fBCTManagerMain.CreateCT();
  IF iNewCt <> 0 THEN 
    LogLvl(Lvl:=E_LogSeverity.Debug, Msg:=F_Concat2('CreateCT: ', TO_STRING(iNewCt.pCT^.iId)));
    pCT := fBCTManagerMain.GetContainerInstance(iCT:=iNewCt);
    IF pCT <> 0 THEN
      pCT^.LogLevel := LogLevel;            // apply module masters logLevel to CTs

      // setup new CT
      iNewCt.bProductPresent := TRUE;
      iNewCt.SetPosX0(nPosDomain:=E_PosDomain.master_pos, nXO:= _iMasterStartPosDetect.nStartPositionX0); 
      iNewCt.SetPosX0(nPosDomain:=E_PosDomain.pos_px,     nXO:= _iMasterStartPosDetect.nStartPositionX0 / FC_LREAL_TO_DINT(_iMasterPos.fSubPxResolution));
      // Production Manger
      _pProdMngr^.CT_Create(sCT := iNewCt); 
      _pProdMngr^.CT_Produce(sCT := iNewCt);   // produce this CT
      // Prepare deformation CT
      pCT^.StartScript(iDeformationHandler:=THIS^); // we do not have a script worker, just start it here
		END_IF
  END_IF
END_IF


fBCTManagerMain.nPositions[E_PosDomain.master_pos] := nMasterPosition;
fBCTManagerMain.nPositions[E_PosDomain.pos_px]     := nMasterPosition/TO_DINT(nC_SubPixelResolution);
fBCTManagerMain();

// view
nViewPmSel := TO_UDINT(LIMIT(1, TO_DINT(nViewPmSel), iCPr_NB_PM));  // limit visu selection

METHOD DeleteCachedCt : BOOL
VAR_INPUT
	iCT	: I_CT;
END_VAR


// nothing to do or later TODO: DeleteCT in CTM?
END_METHOD

(*
  Distance (Offset) from Master-Trigger to Master Reference Position.
  NOTE: This is normally the distance between the first (MASTER) StartPosDetection to first print Module (Printing Unit) 
*)
PROPERTY fDetectToRefPos : LREAL
GET
IF _pMasterModule = 0 THEN RETURN; END_IF

fDetectToRefPos := _pMasterModule^.fDetectToPm;
END_GET
END_PROPERTY

(*Distance from first to last print module*)
PROPERTY fLastModuleOffset : LREAL
GET
fLastModuleOffset := 1;
END_GET
END_PROPERTY

PROPERTY iHardwarePool : I_HardwarePool
GET
iHardwarePool := _iHwPool;
END_GET
END_PROPERTY

PROPERTY iMasterPrintPosition : I_PrintPosition
GET
iMasterPrintPosition := _iMasterPos;
END_GET
END_PROPERTY

METHOD Init : BOOL
VAR_INPUT
  pPU : POINTER TO FB_PU;
  pProdMngr : POINTER TO FB_ProdManager_DMAX;
  iHwPool : I_HardwarePool;
END_VAR
IF pPU = 0 OR pProdMngr = 0 OR iHwPool = 0 THEN LogError('init() invalid init parameter'); RETURN; END_IF

_pPU := pPU;
_pProdMngr := pProdMngr;
_iHwPool := iHwPool;

fBCTManagerMain.Init();

bInit := TRUE;
END_METHOD

PROPERTY iWorkerParams : I_WorkerParams
GET
iWorkerParams := THIS^;
END_GET
END_PROPERTY

PROPERTY pCTManager : POINTER TO FB_CTManagerDefGrid
GET
pCTManager := ADR(fBCTManagerMain);
END_GET
END_PROPERTY

METHOD registerModule : BOOL
VAR_INPUT
  pModule : POINTER TO FB_PrintModule_Base;
END_VAR
IF pModule = 0 THEN LogError('registerModule() invalid module given, ignore'); RETURN; END_IF
IF _nModules >= nC_MaxModules THEN LogError(F_Concat2('registerModule() too many already registered, ignore', pModule^.InstanceName)); RETURN; END_IF

// add new
_nModules := _nModules + 1;
_sModules[_nModules] := pModule;

// set first as master (can be changed again with a call to setMasterModule())
IF _nModules = 1 THEN setMasterModule(pModule:=pModule); END_IF  

registerModule := TRUE;
END_METHOD

(*
  Register for PU StatusClient
*)
METHOD registerPuStatusClient : BOOL
VAR_INPUT
	sClient	: CalmarCompPrint.I_PrintStatusClient;
END_VAR
registerPuStatusClient := _pPU^.registerStatusClient(sClient:=sClient);
END_METHOD

METHOD registerPuSubystem : BOOL
VAR_INPUT
	iSubSys	: I_PrintSubsystem;
END_VAR
_pPU^.registerStatusClient(sClient := iSubSys);
_pPU^.registerSubystem(sSubSys:= iSubSys);
END_METHOD

METHOD setMasterModule : BOOL
VAR_INPUT
  pModule : POINTER TO FB_PrintModule_Base;
END_VAR
VAR
  i : UDINT;
  bFound : BOOL;
END_VAR
// note make this a private method if MasterModule knows it modules
IF pModule = 0 THEN LogError('setMasterModule: invalid module given, ignore'); RETURN; END_IF

// search if module is registered
bFound := FALSE;
FOR i:=1 TO _nModules DO
  IF pModule = _sModules[i] THEN  // found
    bFound := TRUE; EXIT;
	END_IF
END_FOR
IF NOT bFound THEN
  LogError(F_Concat2('Could not set as master module (not registered): ', pModule^.InstanceName)); 
  RETURN; 
END_IF

_pMasterModule := pModule;
END_METHOD

END_FUNCTION_BLOCK

// ---- POUs/Products/Print_Weu/FB_HardwarePool.TcPOU
FUNCTION_BLOCK FB_HardwarePool EXTENDS T_NamedBase IMPLEMENTS I_HardwarePool
VAR_INPUT
END_VAR
VAR_OUTPUT
END_VAR
VAR
  //Registered devices
  _rPc   : ARRAY [1..iCPr_NB_PC] OF POINTER TO FB_PC;
  _rPh   : ARRAY [1..iCPr_NB_PH] OF POINTER TO FB_PH;
  _nPcCount : UDINT;
  _nPhCount : UDINT;
  
  //Initialization data
  _bInitOk             : BOOL;
  _sAmsNetIdLocalhost  : STRING;
  _sAmsNetIdIo         : STRING;
  _pOd                 : POINTER TO FB_OD;        // not yet used (used for intializing pc/pc hardware
  _pConfig             : POINTER TO ST_CONFIG_P;  // not yet used (used for intializing pc/pc hardware
  
  // Firmware update
  (* -- fw/hw upgrade -- *)
  fb_fwhw_update       : FB_CALMAR_UPDATE;
  (* -- hib remote update -- *)
	fb_pc_hib_rupd       : ARRAY[1..iCPr_NB_PC] OF FB_PC_HIB_RUPD;(*HIB remote update channles*)
  fb_hib_rup           : FB_HIB_UPDATE;                         (*HIB remote updater*)
  
  //Visu
  _bVisuInitOk         : BOOL;
  fb_visu_pc                                 : FB_PC_Visu;
  fb_visu_ph                                 : FB_PH_Visu;
  
  fBPcSelector         : FB_VisuSelector;
  fBPhSelector         : FB_VisuSelector;
  
  _rPcVisuSel          : POINTER TO FB_PC;
  _rPhVisuSel          : POINTER TO FB_PH;
  _rAdsPcVisuSel       : POINTER TO ST_ADS_PC;
  _rAdsPhVisuSel       : POINTER TO ST_ADS_PH;
END_VAR

fb_fwhw_update();
fb_hib_rup();

// update visu
visu();

PROPERTY bError_fwhw_update : BOOL
GET
bError_fwhw_update := FALSE;
//bError_fwhw_update := fb_fwhw_update.bL_Upd_Error;
END_GET
END_PROPERTY

PROPERTY bError_hib_rup : BOOL
GET
bError_hib_rup := FALSE;
//bError_hib_rup := fb_hib_rup.bL_Busy;
END_GET
END_PROPERTY

METHOD init
VAR_INPUT
  sAmsNetIdLocalhost  : STRING;
  sAmsNetIdIo         : STRING;
  pOd                 : POINTER TO FB_OD;
  pConfig             : POINTER TO ST_CONFIG_P;
END_VAR
_sAmsNetIdLocalhost  := sAmsNetIdLocalhost;  
_sAmsNetIdIo         := sAmsNetIdIo;         
_pOd                 := pOd;  
_pConfig             := pConfig;



(*File Downloader*)
(*************************************************************************************************)
(* - firmware*)
fb_fwhw_update.aI_appl_file_path := F_Concat3(aC_PlcConfigPath, aC_PlcFlashFileSubPath, 'user.appl');
fb_fwhw_update.aI_fpga_file_path := F_Concat3(aC_PlcConfigPath, aC_PlcFlashFileSubPath, 'user.fpga');
fb_fwhw_update(pI_fbPc:= _rPc);
fb_fwhw_update.init();

(* - hib remote update*)
fb_hib_rup.bI_Enable := TRUE;
fb_hib_rup.aI_FilePath := F_Concat3(aC_PlcConfigPath, aC_PlcFlashFileSubPath, 'user.hib');
fb_hib_rup(sI_Ary_Fb:=fb_pc_hib_rupd, pI_Ary_Fb_Pc:=_rPc);

_bInitOk := TRUE;
END_METHOD

PROPERTY nPcs : UDINT
GET
nPcs := _nPcCount;
END_GET
END_PROPERTY

PROPERTY pPcs : POINTER TO ARRAY[1..iCPr_NB_PC] OF POINTER TO FB_PC
GET
pPcs := ADR(_rPc);
END_GET
END_PROPERTY

METHOD registerPc : BOOL
VAR_INPUT
	pNewPc	    : POINTER TO FB_PC;
END_VAR

VAR
  aName : STRING;
	pAds: INT;
END_VAR
IF _nPcCount<TO_UDINT(iCPr_NB_PC) AND pNewPc <> 0 THEN
  _nPcCount := _nPcCount + 1;
  _rPc[_nPcCount] := pNewPc;
  
  IF _pConfig <> 0 THEN
    (*still done in PRG_PRINT
    aName := _pConfig^.aC_PC_NAME;
    aName :=CONCAT(aName, TO_STRING(_nPcCount)); 
    
    //Init Device
    sNewPc^.init(
      aName               := aName,
      pAdsConfig          := pAdsConfig,
      sAmsNetIdLocalHost  := _sAmsNetIdLocalhost,
      sAmsNetIdIo         := _sAmsNetIdIo,
      nEcatSlaveAddr      := TO_UINT(nC_Pc_EcatBaseAddress+TO_INT(_nPcCount)-1),
      nBlockId            := TO_INT(ePr_BLK_PC),
      pOd                 := _pOd,
      bHeaterEnableExist  := FALSE,
      bPrintEnableExist   := TRUE
   ); *)
  END_IF
ELSE
    LogError('register PC failed');
END_IF
END_METHOD

METHOD registerPh : BOOL
VAR_INPUT
	pNewPh	     : POINTER TO CalmarCompPrint.FB_PH;
  //pAdsConfig   : POINTER TO FB_ADS_Config;
  //pConnectedCb : POINTER TO CalmarCompPrint.FB_PC;
  //iChannel     : INT;
END_VAR

VAR
  aName : STRING;
END_VAR
IF _nPhCount<TO_UDINT(iCPr_NB_PH) AND pNewPh <> 0 THEN
  _nPhCount := _nPhCount + 1;
  _rPh[_nPhCount] := pNewPh;
  
  IF _pConfig <> 0 THEN
    (* still done in PRG_PRINT
    aName := _pConfig^.aC_PH_NAME;
    aName :=CONCAT(aName, TO_STRING(_nPhCount)); 
   
    pNewPh^.init(
      aName              := aName,     
      pAdsConfig         := pAdsConfig,
      sPhDef             := GVL_PrintDef.XAAR_GS12U,    
      tTempMonitor       := T#30S,
      iFoeHandler        := pConnectedCb^,
      iChannel           := iChannel,
      bPositionX_Exist   := TRUE,                               
      aPositionX_Unit    := _pConfig^.aC_PH_POSITION_X_UNIT,   
      lPositionX_Min     := _pConfig^.lL_PH_POSITION_X_SET_MIN, 
      lPositionX_Max     := _pConfig^.lL_PH_POSITION_X_SET_MAX,
      bPositionY_Exist   := TRUE,                              
      aPositionY_Unit    := _pConfig^.aC_PH_POSITION_Y_UNIT,  
      lPositionY_Min     := _pConfig^.lL_PH_POSITION_Y_SET_MIN, 
      lPositionY_Max     := _pConfig^.lL_PH_POSITION_Y_SET_MAX,
      bVoltageScale_Exist := TRUE,
      aVoltageScale_Unit  := '%', 
      fVoltageScale_Min   := 90.0,  
      fVoltageScale_Max   := 110.0 
    );
    *)
  END_IF
ELSE
    LogError('register PH failed');
END_IF
END_METHOD

ACTION visu:
//Init Visu
IF NOT _bVisuInitOk THEN
  fBPcSelector.setAryBounds(iLowerBoundary := 1,iUpperBoundary := TO_DINT(_nPcCount));
  fBPhSelector.setAryBounds(iLowerBoundary := 1,iUpperBoundary := TO_DINT(_nPhCount));
  _bVisuInitOk :=TRUE;
END_IF

//Visu ********************
_rPcVisuSel       := _rPc[fBPcSelector.pSelect^];
_rAdsPcVisuSel    := _rPc[fBPcSelector.pSelect^]^._pAds;
_rPhVisuSel       := _rPh[fBPhSelector.pSelect^];
_rAdsPhVisuSel    := _rPh[fBPhSelector.pSelect^]^._pAdsIf;
END_ACTION

END_FUNCTION_BLOCK

// ---- POUs/Products/Print_Weu/FB_WorkerDefGrid_Inspection.TcPOU
FUNCTION_BLOCK FB_WorkerDefGrid_Inspection EXTENDS FB_WorkerDefGrid
VAR PERSISTENT
  _fWorkerToMasterRef  : LREAL := 3;    (*Distance between Master reference first PM and this worker, mechanisch*)
END_VAR


{warning 'TODO: implement inspection trigger'}

METHOD PROTECTED  Attach : BOOL
VAR_INPUT
  iCT              : I_CT;                         (*container at triggered event position*)
END_VAR
IF SUPER^.Attach(iCT:=iCT) THEN
  ;
END_IF
END_METHOD

PROPERTY fWorkerToMasterRef : LREAL
GET
fWorkerToMasterRef := _fWorkerToMasterRef;
END_GET
END_PROPERTY

METHOD   mJobStart
VAR_INPUT
	sJobDef	: CalmarCompPrint.I_JobDefinition;
END_VAR
END_METHOD

METHOD  mJobStop
VAR_INPUT
	sStatus	: CalmarCompPrint.I_JobStatus;
END_VAR
END_METHOD

METHOD Release : BOOL
VAR_INPUT
  iCT              : I_CT;                         (*container at triggered event position*)
END_VAR
IF SUPER^.Release(iCT := iCT) THEN
  ;  
END_IF
END_METHOD

METHOD  work
SUPER^.work();

//Worker position update
IF _iWorkerParams <> 0 AND _pAttachedCt = 0 THEN     // Update only without attached container
  // WorkerPosition =  Worker<-Master<-CAM<-SheetDetect
  fPosition := _fWorkerToMasterRef + _iWorkerParams.fDetectToRefPos;
END_IF

IF _pAttachedCt <> 0 THEN
  Release(iCT:=_pAttachedCt^);
END_IF
END_METHOD

END_FUNCTION_BLOCK

// ---- POUs/Products/Print_Weu/FB_NeutralFibreDetermine.TcPOU
FUNCTION_BLOCK FB_NeutralFibreDetermine EXTENDS FB_Commons
{library public}
VAR_INPUT
  (*EL1252*)
  bIKp_MarkTrigger01        AT%I* : BOOL;        (*Mark sensor 01*)
  tIKp_TimeStampPos01       AT%I* : T_DCTIME64;  (*TimeStamp Pos_Edge @EL1252*)
  tIKn_TimeStampNeg01       AT%I* : T_DCTIME64;  (*TimeStamp Neg_Edge @EL1252*)
  bIKp_MarkTrigger02        AT%I* : BOOL;        (*Mark sensor 02*)
  tIKp_TimeStampPos02       AT%I* : T_DCTIME64;  (*TimeStamp Pos_Edge @EL1252*)
  tIKn_TimeStampNeg02       AT%I* : T_DCTIME64;  (*TimeStamp Neg_Edge @EL1252*)

  fSpeed                          : LREAL;       (*Current speed of substrate in [m/s]*)
END_VAR

VAR_OUTPUT
END_VAR

(*{library private}*)
VAR
  bInitOk                         : BOOL;           // initialized
  bSpeedValid                     : BOOL;           // speed is valid
  
  (*configuration*)
  _nResolution                    : LREAL := 1;     // Printhead Resolution [e.g. 600] x Subpixel Resolution [e.g. 32]*)

  fbRTrigMark01                   : R_TRIG;
  fbRTrigMark02                   : R_TRIG;
  
  fL_DurationMark01to02           : LREAL;      (*Mark 1 to 2 [ms]*)
  fL_LengthMark01to02             : LREAL;      (*Mark 1 to 2 [mm]*)
  nL_DeltaMark01to02              : DINT;       (*Mark 1 to 2 [SubPx]*)
END_VAR

IF NOT bInitOk THEN RETURN; END_IF;

fbRTrigMark01(CLK := bIKp_MarkTrigger01);
fbRTrigMark02(CLK := bIKp_MarkTrigger02);

IF fbRTrigMark01.Q THEN
	;
END_IF

IF fbRTrigMark02.Q THEN
	fL_DurationMark01to02 := (ULINT_TO_LREAL(tIKp_TimeStampPos02) - ULINT_TO_LREAL(tIKp_TimeStampPos01)) / 1_000_000.0; (*[ms]*)
	fL_LengthMark01to02   := ((fL_DurationMark01to02 / 1000) * fSpeed) * 1000;    (*[mm]*)
	nL_DeltaMark01to02    := LREAL_TO_DINT((fL_LengthMark01to02 * _nResolution) / 25.4);    (*[SubPx]*)
END_IF

(********************************* END OF FB *****************************************************)

METHOD Init
VAR_INPUT
  nResolution                   : LREAL := 1;        (*Printhead Resolution [e.g. 600] x Subpixel Resolution [e.g. 32]*)
END_VAR
(*zero divisions*)
IF nResolution = 0 THEN LogError('Invalid parameter'); RETURN; END_IF;

// configration
_nResolution := nResolution;

bInitOk := TRUE;
END_METHOD

END_FUNCTION_BLOCK

// ---- POUs/Projects/Print/_Test/FB_PrgPrint_test.TcPOU
(*
  Manages the print test/simulation. 
  - It has access to ADS_PU & ADS_Camera & JobManager 
  - It tries to do all the simulation work internally with the given references
  - Else it provides some informations & triggers for external code where this FB has no access to 
*)
FUNCTION_BLOCK FB_PrgPrint_test EXTENDS FB_BasePrint
VAR_OUTPUT
  bO_Power24V_ON  AT%Q* : BOOL;
END_VAR
VAR
  // config
  _pAdsPu : POINTER TO ST_ADS_PU;
  _pAdsSubstrate : POINTER TO ST_ADS_SUBSTRATE;
  _pAdsCamera : POINTER TO ST_ADS_CAMERA;
  
 (*test fb&data instances*)
  fb_JobManagement      : FB_JobManagement;  (*for VISU_JOB_MANAGENT*)


	(*StartUp*)
	cL_DEVS               : UINT := 1;    (*number of test PC devices*)
  
  (*helper*)
  nCtr                  : UDINT;
  sTmpPcFlags           : ST_PC_FLAGS;
  rfTStart, rfTStop     : RF_TRIG;          (*start/stop simulation trigger*)
  rfHwReady, rfTStarting: RF_TRIG;
  rfRunMachine        : RF_TRIG;
  
  _eLogLevel            : E_LogSeverity := E_LogSeverity.Info;
  _bSimPrgPrint, _bMemSimPrgPrint : BOOL;
  _bSimPrgMachine, _bMemSimPrgMachine : BOOL;
  _bSimPrgInk, _bMemSimPrgInk : BOOL;

 
  (*---- script interface ---------------*)
  bHwReady              : BOOL;             (*[status]  hardware is booted and ready (CBs in OP)*)
  bStarting             : BOOL;             (*[status]  test starting*)
  bStopping             : BOOL;             (*[status]  test stopping*)
  bRunning              : BOOL;             (*[status]  simulation runnign*)
  bStart, bStop         : BOOL;             (*[cmd]     start/stop print simulation sequence*)
  bRunMachine           : BOOL;             (*[cmd]     start machine feeder & belt*)

  (*-------------------------------------*)

END_VAR
VAR PERSISTENT
  _bEnTesting            : BOOL;
  _bEnAutoStartPrinting  : BOOL;   // automatically load a job and start printing a test pattern job
  _bEnVerboseMode        : BOOL;
  _bForceHwReady         : BOOL;
  eCameraDevice         : E_CameraDevice := E_CameraDevice.PrintMark;    (*Camera device*)
  eCameraMode           : E_CameraMode := E_CameraMode.Auto;           (*Camera mode*)
  sJobConfig            : ST_JobSettings := (*[cfg]     test job settings*)
  ( // default job
    aI_JobId := '123456780-1111-1111-1111-999999999999',
    lI_StartPage := 1,              // obsolete
    lI_EndPage := 1,                // obsolete
    lI_ImageDepth := 200_000,       // 1_127_082; //[um]
    lI_ImageWidth := 200_000,       // 455_000; //[um]
    lI_ProductionImageCount := 1,
    lI_MaintenanceImageCount := 0,
    lI_NumberOfCopies := 0,
    lI_PrintMode := 16#832200,      // bit set: 9,17,23 (13=endless)
    lI_PrePostBlankDepth := 12361,  // 292px in [um]
    lI_SubPixelResolution := 32,
    lI_ResolutionX := 600,
    aI_JobDescription := 'i1',      // endless p0
    aI_JobName := 'PRG_TEST_job'
  );
END_VAR

IF NOT bInitialized THEN RETURN; END_IF
IF NOT _bEnTesting   THEN RETURN; END_IF

//-- start / stop trigger generation
rfTStart(CLK:=bStart); rfTStop(CLK:=bStop); rfTStarting(CLK:=bStarting); rfHwReady(CLK:=bHwReady); rfRunMachine(CLK:=bRunMachine);

//-- check if hardware is ready
bHwReady := TRUE; 
FOR nCtr := 1 TO TO_UDINT(iCPr_NB_PC) DO
  IF PRG_PRINT.FB_PC[nCtr].bBoardEnable THEN
    sTmpPcFlags := PRG_PRINT.FB_PC[nCtr].sPcFlags;
    IF NOT sTmpPcFlags.bBoardInOp AND NOT _bForceHwReady THEN
      bHwReady := FALSE;
    END_IF 
  END_IF
END_FOR


// auto start stop printing 
IF    _bEnAutoStartPrinting AND rfHwReady.RT THEN bStart := TRUE;
ELSIF _bEnAutoStartPrinting AND rfHwReady.FT THEN bStop := TRUE; 
END_IF 

// starting sequence and status
bStarting := TestStartSequence();
bStopping := TestStopSequence();

// trigger actions
// - update running status
IF rfTStarting.FT THEN bRunning := TRUE;   
ELSIF rfTStop.RT  THEN bRunning := FALSE; END_IF 
// - set debug log level
IF _bEnVerboseMode THEN _eLogLevel := E_LogSeverity.Debug; 
ELSE                    _elogLevel := E_LogSeverity.Info; END_IF

(****  Job Management in ComponentsPrints ****)
fb_JobManagement(pI_Ary_Fb_Pc:= PRG_PRINT.pFB_PC^);

PROPERTY bChangedPrgSim : BOOL
GET
bChangedPrgSim := isPrgSimUpdate();
END_GET
END_PROPERTY

PROPERTY bEnterSim : BOOL
GET
bEnterSim := rfTStart.RT;
END_GET
END_PROPERTY

PROPERTY bEnTesting : BOOL
GET
bEnTesting := _bEnTesting;
END_GET
SET
_bEnTesting := bEnTesting;
END_SET
END_PROPERTY

PROPERTY bExitSim : BOOL
GET
bExitSim := rfTStop.RT;
END_GET
END_PROPERTY

PROPERTY bSimPrgInk : BOOL
GET
bSimPrgInk := _bSimPrgInk;
END_GET
SET
_bSimPrgInk := bSimPrgInk;
END_SET
END_PROPERTY

PROPERTY bSimPrgMachine : BOOL
GET
bSimPrgMachine := _bSimPrgMachine;
END_GET
SET
_bSimPrgMachine := bSimPrgMachine;
END_SET
END_PROPERTY

PROPERTY bSimPrgPrint : BOOL
GET
bSimPrgPrint := _bSimPrgPrint;
END_GET
SET
_bSimPrgPrint := bSimPrgPrint;
END_SET
END_PROPERTY

PROPERTY bStartMachine : BOOL
GET
bStartMachine := rfRunMachine.RT;
END_GET
END_PROPERTY

PROPERTY bStopMachine : BOOL
GET
bStopMachine := rfRunMachine.FT;
END_GET
END_PROPERTY

METHOD Init : BOOL
VAR_INPUT
  pAdsPu  : POINTER TO ST_ADS_PU;
  pAdsCamera : POINTER TO ST_ADS_CAMERA;
  pAdsSubstrate : POINTER TO ST_ADS_SUBSTRATE;
END_VAR
IF pAdsPu = 0 OR pAdsCamera = 0 OR pAdsSubstrate = 0 THEN
  LogError('Invalid init parameter');
  RETURN;
END_IF

_pAdsPu := pAdsPu;
_pAdsCamera := pAdsCamera;
_pAdsSubstrate := pAdsSubstrate;

(*init JobManager*)
// or default job // sJobConfig := fb_JobManagement.getJobSettings();
fb_JobManagement.Init(pI_JobSettings:=ADR(sJobConfig));

bInitialized := TRUE;
END_METHOD

METHOD isLogLevelUpdate : BOOL
VAR_OUTPUT
  eLogSeverity : E_LogSeverity;
END_VAR
VAR_INST
  oldLogSeverity : E_LogSeverity := E_LogSeverity.Info;
END_VAR
isLogLevelUpdate := SEL(oldLogSeverity <> _eLogLevel, FALSE, TRUE);
oldLogSeverity := _eLogLevel;     // remember level

eLogSeverity := _eLogLevel;
END_METHOD

METHOD PRIVATE isPrgSimUpdate : BOOL
VAR
  bChange : BOOL;
END_VAR
IF _bSimPrgInk     <> _bMemSimPrgInk     THEN _bMemSimPrgInk     := _bSimPrgInk;     bChange := TRUE; END_IF
IF _bSimPrgMachine <> _bMemSimPrgMachine THEN _bMemSimPrgMachine := _bSimPrgMachine; bChange := TRUE; END_IF
IF _bSimPrgPrint   <> _bMemSimPrgPrint   THEN _bMemSimPrgPrint   := _bSimPrgPrint;   bChange := TRUE; END_IF

isPrgSimUpdate := bChange;
END_METHOD

(*
  Load a test job
  :return: TRUE as long command is busy
*)
METHOD LoadTestJob : BOOL
VAR_INPUT
  bLoad : BOOL; 
END_VAR
VAR_INST
  bBusy : BOOL;
  tLoadTimeout : TIME;
  tExecute : TON := (PT:=T#20S);
END_VAR
IF NOT bLoad OR tExecute.Q THEN  // disable or timeout -> abort
  tExecute(IN:=FALSE);
  LoadTestJob := bBusy := FALSE;
  RETURN;
END_IF

tLoadTimeout := TO_TIME((sJobConfig.lI_ImageWidth/1000)*(sJobConfig.lI_ImageDepth/1000));             // (w[mm] * d[mm])/1000 = [s] 

tExecute(IN:=bLoad, PT:=SEL(_bForceHwReady, tLoadTimeout, T#4S));
IF NOT bBusy THEN
  // - load job
  fb_JobManagement.LoadJob(aI_AmsNetId_Io:=sC_AMSNETID_IO, pI_JobSettings:=ADR(sJobConfig));
  
  // - setup PU job
  _pAdsPu^.sI_JobSettings := sJobConfig;
  
  bBusy := TRUE;
ELSE
  bBusy := fb_JobManagement.bO_Busy; 
END_IF

LoadTestJob := bBusy;
END_METHOD

METHOD StartJob : BOOL
VAR_INPUT
END_VAR
VAR_INST
  bBusy : BOOL;
END_VAR
IF NOT _pAdsPu^.sI_Start.bI_Command THEN
  _pAdsPu^.sI_Start.bI_Command := TRUE;
  bBusy := TRUE;
ELSE    
  _pAdsPu^.sI_Start.bI_Command := FALSE;
  bBusy := FALSE;
END_IF

StartJob := bBusy;
END_METHOD

METHOD PRIVATE StopJob : BOOL
VAR_INPUT
END_VAR
VAR_INST
  bBusy : BOOL;
END_VAR
IF NOT _pAdsPu^.sI_Stop.bI_Command THEN
  _pAdsPu^.sI_Stop.bI_Command := TRUE;
  bBusy := TRUE;
ELSE    
  _pAdsPu^.sI_Stop.bI_Command := FALSE;
  bBusy := FALSE;
END_IF

StopJob := bBusy;
END_METHOD

(*
  :return: TRUE if busy
*)
METHOD PRIVATE TestStartSequence : BOOL
VAR_INPUT
END_VAR
VAR_INST
  nState			    : INT := 0;     (*start-up fsm state variable*)
  nNumDevices     : UINT;         (*loop variable*)
  nExtPcSelector  : DINT;
  tWaitJobStart   : TON := (PT:=T#4S);  (*Wait before starting job (generate pattern job)*)
END_VAR
(*-------------------------------------------*)
(* This initialize all necessary modules prior to test start*)

(*Setup Testing VarData*)
CASE nState OF

(*======> Start and Init*)
0: (*--- IDLE/START ---*)
  IF bStart THEN
    // prepare job downloader
    nNumDevices := cL_DEVS;   // set number of pc devices
    fb_JobManagement.setExtSelect(pI_Selector:=ADR(nExtPcSelector));
    nState := 1;
	END_IF

1: (*--- enter module simulations ---*)
  _bSimPrgPrint         := TRUE;
  _bSimPrgMachine       := TRUE;
  _bSimPrgInk           := TRUE;
  //_bEnVerboseMode       := TRUE;
  bO_Power24V_ON        := TRUE;
  nState := 10;
  

10: (*--- Started ---*)
  IF bStart OR nNumDevices > 0 THEN
    nState := 11;
    nExtPcSelector := nNumDevices;
  END_IF

(*======> Load initial job*)
11: (*start load default job and wait until not busy*)
  IF bHwReady OR _bForceHwReady THEN
    nState := 12;
  END_IF
  
12: (*start load default job and wait until not busy*)
  IF NOT LoadTestJob(bLoad:=TRUE) THEN 
    nNumDevices := nNumDevices - 1;
    IF nNumDevices > 0 THEN
      nState := 10;
    ELSE
      nState := 30;
    END_IF
  END_IF

(*=======> command PRG_PRINT*)
30: (*--- write job settings ---*)
  IF NOT WriteJobSettings() THEN
    nState := 40;
    tWaitJobStart(IN:=FALSE); // reset timer
    tWaitJobStart(IN:=TRUE);
  END_IF

40: (*--- wait for job generated/loaded ---*)
  IF tWaitJobStart.Q THEN
    tWaitJobStart(IN:=FALSE);
    nState := 50;
  END_IF

50: (*--- start Job ---*)
  IF NOT StartJob() THEN
    tWaitJobStart(IN:=FALSE); // reset timer
    tWaitJobStart(IN:=TRUE);
    nState := 60;
  END_IF

60: (*--- Wait for job started ---*)
  IF tWaitJobStart.Q THEN
    tWaitJobStart(IN:=FALSE);
    bRunMachine     := TRUE;            // start machine
    nState := 99;
	END_IF

98: (*Error*)
  nState := 99;

99: (*Done*)
  bStart := FALSE;
  nState := 0;

END_CASE

tWaitJobStart();
TestStartSequence := SEL(nState=0, TRUE, FALSE);
END_METHOD

(*
  :return: TRUE if busy
*)
METHOD PRIVATE TestStopSequence : BOOL
VAR_INPUT
END_VAR
VAR_INST
  nState			    : INT := 0;     (*start-up fsm state variable*)
  nNumDevices     : UINT;         (*loop variable*)
  nExtPcSelector  : DINT;
END_VAR
(*-------------------------------------------*)
(* This initialize all necessary modules prior to test start*)

(*Setup Testing VarData*)
CASE nState OF

(*======> Start and Init*)
0: (*--- IDLE/START ---*)
  IF bStop THEN
    bRunMachine := FALSE;
    //
    nNumDevices := cL_DEVS;   // set number of pc devices
    fb_JobManagement.setExtSelect(pI_Selector:=ADR(nExtPcSelector));
    nState := 1;
	END_IF

1: (*--- Started ---*)
  IF bStop OR nNumDevices > 0 THEN
    nState := 10;
    nExtPcSelector := nNumDevices;
  END_IF
  
10: (*--- for all CB ---*)
  nNumDevices := nNumDevices - 1;
  bStart := FALSE;
  IF nNumDevices > 0 THEN
    nState := 1;
  ELSE
    nState := 20;
  END_IF
  
(*======> Load initial job*)
20: (*stop job*)
  IF NOT StopJob() THEN
    nState := 60;
  END_IF
  
60: (*--- enter module simulations ---*)
  _bSimPrgPrint         := FALSE;
  _bSimPrgMachine       := FALSE;
  _bSimPrgInk           := FALSE;
  _bEnVerboseMode       := FALSE;
  bO_Power24V_ON        := FALSE;
  nState := 99;

98: (*Error*)
  nState := 99;

99: (*Done*)
  bStop := FALSE;
  nState := 0;

END_CASE

TestStopSequence := SEL(nState=0, TRUE, FALSE);
END_METHOD

(*
  :return: TRUE if busy
*)
METHOD PRIVATE WriteJobSettings : BOOL
VAR_INPUT
END_VAR

_pAdsPU^.sI_JobSettings := sJobConfig;  // set internal job settings to ads

//_pAdsSubstrate^.sI_SizeX.fI_Val := TO_REAL(sJobConfig.lI_ImageDepth);
//_pAdsSubstrate^.sI_SizeY.fI_Val := TO_REAL(sJobConfig.lI_ImageWidth);

// - setup Camera 
_pAdsCamera^.eI_CameraDevice := eCameraDevice;
_pAdsCamera^.eI_CameraMode   := eCameraMode;
//_pAdsCamera^.eI_CameraDevice := eCameraDevice; // set camera selection
//_pAdsCamera^.eI_CameraMode := eCameraMode;

// - setup substrate
_pAdsSubstrate^.aI_SubstrateName := 'A TestSubtrate equal to image dimension';
_pAdsSubstrate^.sI_SizeX.fI_Val := TO_REAL(_pAdsPu^.sI_JobSettings.lI_ImageDepth) / 1_000;  // [um] -> [mm]
_pAdsSubstrate^.sI_SizeY.fI_Val := TO_REAL(_pAdsPu^.sI_JobSettings.lI_ImageWidth) / 1_000;  // [um] -> [mm]
_pAdsSubstrate^.sI_SizeZ.fI_Val := 0;

WriteJobSettings := FALSE;
END_METHOD

END_FUNCTION_BLOCK

// ---- POUs/Projects/Print/_Test/PRG_TEST.TcPOU
PROGRAM PRG_TEST
(*************************************************************************************************)
(*  FILENAME:    PRG_TEST.EXP                                                                    *)
(*  PROJECT:     CALMAR PUPLC                                                                    *)
(*  COPYRIGHT:   All rights reserved (c) Wifag//Polytype, Fribourg/Switzerland (2016)            *)
(*  ENVIRONMENT: TwinCAT PLC                                                                     *)
(*  VERSION:     <version>                                                                       *)
(*************************************************************************************************)
(*  DESCRIPTION:                                                                   <description> *)
(*    Controls the test functions.                                                               *)
(*                                                                                </description> *)
(*************************************************************************************************)

VAR
	bL_FirstRun           : BOOL := TRUE;

  (*Test CONFIGURATION*)
  bLogRateKill : BOOL;
  tLog : TON;
  nLogCt : UDINT;
END_VAR

(* INIT First action init call*)
IF bL_FirstRun THEN
	bL_FirstRun := FALSE;
	Init();
END_IF;

(*** configure tests ****************************)
(*--> un-comment the defines in GVL_TestCfg*)
(************************************************)

IF bLogRateKill THEN
  tLog(IN:=NOT tLog.Q, PT:=T#10MS);
  nLogCt := nLogCt + 1;
  F_LogWarning(F_Concat2('LogKill ct: ', TO_STRING(nLogCt)));
END_IF

(*** Library testing ***)
{IF defined (variable: GVL_TestCfg.do_LibTest)}
  LibTest();
{END_IF}

ACTION Init:

; // nothing to do
END_ACTION

ACTION LibTest:
CalmarCommons.PRG_TEST();
CalmarCompPrint.PRG_TEST();
END_ACTION

END_PROGRAM

// ---- POUs/Projects/System/PRG_SYSTEM.TcPOU
PROGRAM PRG_SYSTEM
(*************************************************************************************************)
(*  FILENAME:    PRG_SYSTEM.EXP                                                                  *)
(*  PROJECT:     CALMAR PUPLC                                                                    *)
(*  COPYRIGHT:   All rights reserved (c) Wifag//Polytype, Fribourg/Switzerland (2016)            *)
(*  ENVIRONMENT: TwinCAT PLC                                                                     *)
(*  VERSION:     <version>                                                                       *)
(*************************************************************************************************)
(*  DESCRIPTION:                                                                   <description> *)
(*    Controls the system functionalities.                                                       *)
(*    Main functions: register the module blocks, ADS block generation, ADS module mapping.      *)
(*                                                                                </description> *)
(*************************************************************************************************)
VAR
  bL_InitOK                  : BOOL := FALSE;
  
  sC_Ads_Info                : ST_ADS_INFO;
  sC_Ads_System              : ST_ADS_SYSTEM;
  ISystemBase                : I_SystemBase;                // reference to system base
  
  // Message control
  nMsgResetRequests          : UINT;
  fb_RTrigMsgResetRequest    : R_TRIG;
  
  // Version
  stProgramVersion           : ST_LibVersion;               // version information of project from TwinCAT dialog entry
  aCurrentDateTime           : STRING;  
  
  // View
  nMainVisuFrameIndex        : UINT := 0;   // VISU_Main frame selection
  sMainButtons               : ARRAY[0..4] OF ST_ButtonFrameSel_Def := [
                                                (sImgId:='droplet_w',   nFrameIdx:=0, pFrameSelect:=ADR(nMainVisuFrameIndex), sVisuName:='InkSystem'),
                                                (sImgId:='printer_w',   nFrameIdx:=1, pFrameSelect:=ADR(nMainVisuFrameIndex), sVisuName:='Print'),
                                                (sImgId:='book_w',      nFrameIdx:=2, pFrameSelect:=ADR(nMainVisuFrameIndex), sVisuName:='Recipe'),
                                                (sImgId:='gear_w',      nFrameIdx:=3, pFrameSelect:=ADR(nMainVisuFrameIndex), sVisuName:='Service'),
                                                (sImgId:='lightning_w', nFrameIdx:=4, pFrameSelect:=ADR(nMainVisuFrameIndex), sVisuName:='Machine')
                                              ];
END_VAR

// Init
IF NOT bL_InitOK THEN Init(); END_IF;

(* Message control
  Some errors in the PLC needs TO reset twice TO clear the error completely.
  Message reset from Gallus will be send twice to the PUC.
*)
{warning 'TODO: test if msg reset still works'}
fb_RTrigMsgResetRequest(CLK := PRG_MACHINE.IbEAP_MessageReset);
IF fb_RTrigMsgResetRequest.Q THEN nMsgResetRequests := 2; END_IF
IF nMsgResetRequests > 0 THEN
  IF NOT PRG_SYSTEMBASE.resetPucMessages() THEN
    // request done
    nMsgResetRequests := nMsgResetRequests - 1;
	END_IF
END_IF

(*Get current time*)
aCurrentDateTime := F_Concat3(F_TimeGetDate(), ' ', F_TimeGetTime()); 

(*Call system base*)
PRG_SYSTEMBASE();
PRG_MACHINE.updateSleepLock(); // must be called after SystemBase, to overwrite CanEx

METHOD Init
(*--- init call only once*)
IF bL_InitOK = TRUE THEN RETURN; END_IF

// Get system reference
ISystemBase := PRG_SYSTEMBASE.getSystemBaseInterface();
IF ISystemBase = 0 THEN RETURN; END_IF
// Wait until system(base) is booted
IF ISystemBase.bBooting THEN RETURN; END_IF


// System specific setup
sC_Ads_System.aMachine        := aC_NAME_PRODUCT;
sC_Ads_System.aProject        := aC_NAME_PROJECT;
sC_Ads_System.aProjectVersion := aC_VERSION_PRODUCT;
sC_Ads_System.iVersion        := iC_VERSION_PRODUCT;

// module specific setup
PRG_SYSTEMBASE.setup( pI_Ads_Info               := ADR(sC_Ads_Info)
                    , pI_Ads_System             := ADR(sC_Ads_System));
// --> done in PRG_SYSTEMBASE



//PRG_SYSTEMBASE.sI_AppInfo := _AppInfo;
IF F_CmpLibVersion(stLibVersion_CalmarCompSystem, 1, 6, 1, 0) < 0 THEN
  // because of FB_Maintenance and used template visu in VISU_SYSTEM
  F_Log(LogSeverity:=E_LogSeverity.Error, 'PRG_SYSTEMBASE requires CalmarCompSystem >= 1.6.1');
END_IF

(*--- set library and project versions*)
PRG_SYSTEMBASE.SetVersion(aI_Name:='Tc2_System', stLibVersion_Tc2_System);

stProgramVersion := F_GetVersion();
stProgramVersion.sVersion := F_BuildVersionString(F_GetVersion());
PRG_SYSTEMBASE.SetVersion(aI_Name:='PlcProject', stProgramVersion);

{IF defined (variable: stLibVersion_CalmarCommons)}
  PRG_SYSTEMBASE.SetVersion(aI_Name:='CalmarCommons', stLibVersion_CalmarCommons);
{END_IF}
{IF defined (variable: stLibVersion_CalmarCompDevices)}
  PRG_SYSTEMBASE.SetVersion(aI_Name:='CalmarCompDevices', stLibVersion_CalmarCompDevices);
{END_IF}
{IF defined (variable: stLibVersion_CalmarCompSystem)}
  PRG_SYSTEMBASE.SetVersion(aI_Name:='CalmarCompSystem', stLibVersion_CalmarCompSystem);
{END_IF}
{IF defined (variable: stLibVersion_CalmarCompPrint)}
  PRG_SYSTEMBASE.SetVersion(aI_Name:='CalmarCompPrint', stLibVersion_CalmarCompPrint);
{END_IF}
{IF defined (variable: stLibVersion_CalmarCompMachine)}
  PRG_SYSTEMBASE.SetVersion(aI_Name:='CalmarCompMachine', stLibVersion_CalmarCompMachine);
{END_IF}
{IF defined (variable: stLibVersion_CalmarCompInkSystem)}
  PRG_SYSTEMBASE.SetVersion(aI_Name:='CalmarCompInk', stLibVersion_CalmarCompInkSystem);
{END_IF}
{IF defined (variable: stLibVersion_CalmarCompTcpIp)}
  PRG_SYSTEMBASE.SetVersion(aI_Name:='CalmarCompTcpIp', stLibVersion_CalmarCompTcpIp);
{END_IF}
{IF defined (variable: stLibVersion_CalmarProdDmax)}
  PRG_SYSTEMBASE.SetVersion(aI_Name:='CalmarProdDmax', stLibVersion_CalmarProdDmax);
{END_IF}


(*--- done*)
bL_InitOK := TRUE;
END_METHOD

END_PROGRAM

// ---- Project Information/F_GetVersion.TcPOU
// This function has been automatically generated from the project information.
{attribute 'signature_flag' := '1073741824'}
{attribute 'TcGenerated'}
{attribute 'no-analysis'}
FUNCTION F_GetVersion : ST_LibVersion
VAR_INPUT
	
END_VAR

F_GetVersion.iMajor := 1;
F_GetVersion.iMinor := 1;
F_GetVersion.iBuild := 0;
F_GetVersion.iRevision := 0;
F_GetVersion.sVersion := '1.1.0';
F_GetVersion.nFlags := 0;

END_FUNCTION

// ---- POUs/CheckBounds.TcPOU
// Implicitly generated code : DO NOT EDIT
FUNCTION CheckBounds : DINT
(*************************************************************************************************)
(*  FILENAME:    CHECKBOUNDS.EXP                                                                 *)
(*  PROJECT:     CALMAR PUPLC                                                                    *)
(*  COPYRIGHT:   All rights reserved (c) Wifag//Polytype, Fribourg/Switzerland (2016)            *)
(*  ENVIRONMENT: TwinCAT PLC                                                                     *)
(*  VERSION:     <version>                                                                       *)
(*************************************************************************************************)
(*  DESCRIPTION:                                                                   <description> *)
(*     This function checks `index` with the limits `lower` and `upper`.                         *)
(*     If the limits are exceeded the value is set to the limit and returned by this FC.         *)
(*     In case of a conversion error the debug counter `PRG_SYSTEM.lI_BoundsErr` will be sum up. *)
(*                                                                                </description> *)
(*************************************************************************************************)

VAR_INPUT
	index, lower, upper: DINT;
END_VAR

// Implicitly generated code : Only an Implementation suggestion
{noflow}
IF  index < lower THEN
  CheckBounds := lower;
  F_Report_Error(ErrType:=EN_REPORT_ERROR_TYPE.Report_Error_Bounds);
ELSIF  index > upper THEN
  CheckBounds := upper;
  F_Report_Error(ErrType:=EN_REPORT_ERROR_TYPE.Report_Error_Bounds);
ELSE  
  CheckBounds := index;
END_IF
{flow}

END_FUNCTION

// ---- POUs/CheckPointer.TcPOU
// Implicitly generated code : DO NOT EDIT
FUNCTION CheckPointer : POINTER TO BYTE
VAR_INPUT 
	ptToTest : POINTER TO BYTE; // Destination address of the pointer
	iSize : DINT;		        // Size of the type the pointer points to. (e.g: 20 for POINTER TO ARRAY [0..9] OF INT) 
	iGran : DINT;		        // Granularity of the pointer access. This is the size of the biggest non-structured data type in the type the pointer points to. (e.g: 2 for POINTER TO ARRAY [0..9] OF INT)
	bWrite: BOOL;		        // Indicates read or write Access. TRUE = write access.
END_VAR

IF ptToTest=0 THEN
    ADSLOGSTR(ADSLOG_MSGTYPE_ERROR OR ADSLOG_MSGTYPE_STRING,'CheckPointer failed due to invalid destination address.','');
ELSIF iSize<=0 THEN
    ADSLOGSTR(ADSLOG_MSGTYPE_ERROR OR ADSLOG_MSGTYPE_STRING,'CheckPointer failed due to invalid size.','');
ELSIF iGran<=0 THEN
    ADSLOGSTR(ADSLOG_MSGTYPE_ERROR OR ADSLOG_MSGTYPE_STRING,'CheckPointer failed due to invalid granularity.','');
// -> Please note that the following memory area check is time consuming:
//ELSIF F_CheckMemoryArea(pData:=ptToTest,nSize:=DINT_TO_UDINT(iSize)) = E_TcMemoryArea.Unknown THEN
//    ADSLOGSTR(ADSLOG_MSGTYPE_ERROR OR ADSLOG_MSGTYPE_STRING,'CheckPointer failed due to unknown memory area.','');
END_IF
CheckPointer := ptToTest;
{flow}

END_FUNCTION

// ---- POUs/Products/FB_InspectionSystemTrigger.TcPOU
(*
    Generate timestamp trigger output based on timestamp sensor input. Two variants    
    exist, a timebased approach where the trigger time is calculated at the time the sensor
    event occurs, and a second approach where the sensor event time is translated to a sensor
    event position, and a trigger is generated when the calculated trigger position has almost 
    been reached. The second approach has the advantage that is is less susceptible to speed
    variations.
*)
FUNCTION_BLOCK FB_InspectionSystemTrigger EXTENDS FB_Commons
{library PUBLIC}
VAR_INPUT
  (*System signals*)
  bI_SensorState                  : BOOL;                   // Sensor signal
  (*used if _bUsePositionTrigger = TRUE*)
  iI_CurrentPos                   : DINT;                   // Current position in [SubPx]
  fI_ConveyorSpeed                : LREAL;                  // Current speed of substrate in [m/s]
  iI_SensorX0                     : DINT;                   // Detected X0 position of sensor [SubPx]
  (*used if _bUsePositionTrigger = FALSE*)
  tI_SensorTimeStampPos           : T_DCTIME64;             // Sensor last detection timestamp
  
  (*Debug & Test*)
  bI_ManualTrigger                : BOOL;                   // Manual start trigger
END_VAR

VAR_OUTPUT
  (*Link to EL2252*)
  ObTrigger                 AT%Q* : BOOL;                   // EL2252 Output1 - TRUE=start camer
  OtTriggerStartTime        AT%Q* : T_DCTIME64;             // EL2252 Timestamp - where to set outputs
  OnTriggerCommand          AT%Q* : BYTE;                   // EL2252 Command - activation timestamp ouput
END_VAR

(*{library private}*)
VAR
  bInitOk                         : BOOL;           // initialized
  bSpeedValid                     : BOOL;           // speed is valid
  bTriggerArmed                   : BOOL;           // trigger is armed
  rT_Sensor                       : R_TRIG;         // rising edge trigger sensor
  
  (*configuration*)
  _nResolution                    : LREAL := 1;     // Printhead Resolution [e.g. 600] x Subpixel Resolution [e.g. 32]*)
  _bUsePositionTrigger            : BOOL;           // FALSE: Calculate time with speed and position distance@sensor event, TRUE: Calculate sensor event position, launch trigger based on position
  _fTriggerLength                 : LREAL := 10;    // Length of trigger signal in ms, min. 3 bus cycles
  
 
  eState                          : BYTE;            (*State*)
  tSensor_TimeStamp               : T_DCTIME64;      (*Sensor last detection timestamp*)
  tCurrentTime                    : T_DCTIME64;      (*Current system dc time [64bit]*)
  tTrigger_EventTime              : T_DCTIME64;      (*Trigger event timestamp*)

  _bManualStart                   : BOOL;
  fDeltaDistance                  : LREAL;           (*Distance that the substrate moved between the detection and the treatment of the information [m]*)
  _nX0                            : DINT;            (*Detected X0 position of CT [SubPx] by sensor*)
  _nCamStartPos                   : DINT;            (*Camera start position*)
  _nCamStartedPos                 : DINT;            (*Camera started position [SubPx]*)
  
  tCurrentTimeStamp               : T_DCTIME64;      (* Get Current Timestamp *)
  tLastTimeStamp                  : T_DCTIME64;      (* Get Current Timestamp *)
  fCycleTime                      : LREAL;           (* Current calcualted cycle time [s]*)

  fRemDist                        : LREAL;           (*Remaining distance until trigger occurs [m]*)
  fPreTriggerPosition             : LREAL;           (*Margin between effective trigger position and generation of timestamp*)

  fb_FTrig_ManualTeach            : F_TRIG;          (*FTrig for teach to release inhibit*)
  
  (*Debug*)
  _bVerbose                       : BOOL;
END_VAR

VAR CONSTANT
  fC_MIN_CONVEYOR_SPEED           : LREAL := 0.01;
  fC_PreTrigFactor                : LREAL := 3.0;
  fC_SheetLengthMargin            : LREAL := 0.01;   (*Added 10 mm margin for substrate length in case of print quality strips at the end of sheet in case of start with edge*)

  (*State*)
  cL_IDLE                         : BYTE := 0;       (*Idle state, no trigger active*)
  cL_SENSOREVENT                  : BYTE := 1;       (*Sensor started trigger generation*)
  cL_WAITALMOSTSTART              : BYTE := 2;       (*Wait timestamp calculation critera*)
  cL_WAITSTART                    : BYTE := 3;       (*Wait for trigger generation critera*)
  cL_WAITFEEDBACK                 : BYTE := 4;       (*Wait on feedback from trigger*)
  cL_TRIGACTIVE                   : BYTE := 5;       (*Trigger set*)
  cL_WAITSTOP                     : BYTE := 6;       (*Trigger reset*)

  (*EL2252 Command*)
  cL_INACTIVE                     : BYTE := 0;
  cL_ACTIVE                       : BYTE := 3;
END_VAR

VAR PERSISTENT
  bR_Enable                       : BOOL  := TRUE;   (*Enable system*)
  fR_DeltaDistance                : LREAL := 0.010;  (*Distance that the substrate moved between the detection and the treatment of the information [m]*)
  nR_TimeDistance                 : ULINT := 50;     (*Time that the substrate moved between the detection and the treatment of the information [ms]*)
END_VAR

IF NOT bInitOk THEN RETURN; END_IF;

// General calculations
bSpeedValid   := fI_ConveyorSpeed > fC_MIN_CONVEYOR_SPEED;    // speed valid (ignore trigger if not moving)
tCurrentTime  := F_GetCurDcTaskTime64();                      // current dc time (most accurate time stamp we have)
fCycleTime    := (TO_LREAL(tCurrentTime) - TO_LREAL(tLastTimeStamp)) * 1E-9;  tLastTimeStamp  := tCurrentTime;  // calculate cycle time of this block
bTriggerArmed := bR_Enable AND (bSpeedValid OR NOT _bUsePositionTrigger);

rT_Sensor(CLK := bI_SensorState);

IF NOT bTriggerArmed THEN
  eState := cL_IDLE;
END_IF

(*State Machine ----------------------------------------------------------------*)
CASE eState OF
  cL_IDLE:     (*Not started, waiting for start trigger*)
  
    IF bTriggerArmed THEN (*ignore trigger else*)
       IF rT_Sensor.Q THEN      (*Start launched*)
        eState            := cL_SENSOREVENT;
        tSensor_TimeStamp := tI_SensorTimeStampPos;
        _bManualStart     := FALSE;
      ELSIF bI_ManualTrigger THEN  (*Manual start launched*)
        eState            := cL_SENSOREVENT;
        tSensor_TimeStamp := tCurrentTime;
        _bManualStart     := TRUE;
      END_IF;
    END_IF
    
    OnTriggerCommand := cL_INACTIVE;
    ObTrigger        := FALSE;

  cL_SENSOREVENT:     (*Not started*)
    IF NOT bSpeedValid AND _bUsePositionTrigger THEN 
      eState := cL_IDLE;        // ignore trigger if not moving anymore (avoid zero division)
    ELSE
      (*Position where the sensor has been detected in [SubPx]*)
      _nX0 := iI_SensorX0;
      
      IF _bUsePositionTrigger THEN
        eState             := cL_WAITALMOSTSTART;
      ELSE
        eState             := cL_WAITSTART;
        tTrigger_EventTime := (tSensor_TimeStamp + (nR_TimeDistance * 1_000_000));  (*[ms] to [ns]*)
      END_IF;
      
      OnTriggerCommand := cL_INACTIVE;
      ObTrigger        := TRUE;
    END_IF

  cL_WAITALMOSTSTART: (*Only active when bI_UsePositionTrigger=TRUE: wait until Start position almost reached, then set timestamp*)
    (*Remaining distance in [m], converted to REAL to avoid integer wrap problems*)
    fRemDist             := fR_DeltaDistance + (DINT_TO_LREAL(_nX0) - DINT_TO_LREAL(iI_CurrentPos)) * 0.0254 / _nResolution;
    fPreTriggerPosition  := fC_PreTrigFactor * fCycleTime * fI_ConveyorSpeed;

